LIN {X 0,Y 144.366,Z 912.436,A -85,B 0,C 180,E1 -24295.812,E2 -24295.812} C_VEL
LIN {X 0,Y 143.347,Z 905.875,A -85,B 0,C 180,E1 -24300,E2 -24300} C_VEL
LIN {X 0,Y 143.086,Z 898.213,A -85,B 0,C 180,E1 -24304.225,E2 -24304.225} C_VEL
LIN {X 0,Y 143.586,Z 889.005,A -85,B 0,C 180,E1 -24308.444,E2 -24308.444} C_VEL
LIN {X 0,Y 144.189,Z 880.732,A -85,B 0,C 180,E1 -24311.69,E2 -24311.69} C_VEL
LIN {X 0,Y 145.104,Z 871.718,A -85,B 0,C 180,E1 -24314.731,E2 -24314.731} C_VEL
LIN {X 0,Y 146.264,Z 860.917,A -85,B 0,C 180,E1 -24317.838,E2 -24317.838} C_VEL
LIN {X 0,Y 147.179,Z 852.291,A -85,B 0,C 180,E1 -24319.888,E2 -24319.888} C_VEL
LIN {X 0,Y 144.802,Z 841.839,A -85,B 0,C 180,E1 -24322.072,E2 -24322.072} C_VEL
LIN {X 0,Y 143.37,Z 834.62,A -85,B 0,C 180,E1 -24323.471,E2 -24323.471} C_VEL
LIN {X 0,Y 143.093,Z 834.654,A -85,B 0,C 180,E1 -24329.416,E2 -24329.416} C_VEL
LIN {X 0,Y 143.174,Z 834.808,A -85,B 0,C 180,E1 -24331.231,E2 -24331.231} C_VEL
LIN {X 0,Y 144.079,Z 837.334,A -85,B 0,C 180,E1 -24332.347,E2 -24332.347} C_VEL
LIN {X 0,Y 146.065,Z 839.541,A -85,B 0,C 180,E1 -24334.066,E2 -24334.066} C_VEL
LIN {X 0,Y 146.807,Z 840.16,A -85,B 0,C 180,E1 -24334.663,E2 -24334.663} C_VEL
LIN {X 0,Y 147.849,Z 842.508,A -85,B 0,C 180,E1 -24335.779,E2 -24335.779} C_VEL
LIN {X 0,Y 149.912,Z 845.217,A -85,B 0,C 180,E1 -24337.55,E2 -24337.55} C_VEL
LIN {X 0,Y 154.716,Z 853.873,A -85,B 0,C 180,E1 -24342.069,E2 -24342.069} C_VEL
LIN {X 0,Y 157.954,Z 860.834,A -85,B 0,C 180,E1 -24345.391,E2 -24345.391} C_VEL
LIN {X 0,Y 160.948,Z 868.94,A -85,B 0,C 180,E1 -24349.076,E2 -24349.076} C_VEL
LIN {X 0,Y 163.181,Z 877.591,A -85,B 0,C 180,E1 -24352.913,E2 -24352.913} C_VEL
LIN {X 0,Y 164.31,Z 884.842,A -85,B 0,C 180,E1 -24356.212,E2 -24356.212} C_VEL
LIN {X 0,Y 164.227,Z 886.502,A -85,B 0,C 180,E1 -24356.928,E2 -24356.928} C_VEL
LIN {X 0,Y 160.56,Z 894.538,A -85,B 0,C 180,E1 -24359.772,E2 -24359.772} C_VEL
LIN {X 0,Y 157.298,Z 901.182,A -85,B 0,C 180,E1 -24362.739,E2 -24362.739} C_VEL
LIN {X 0,Y 153.469,Z 908.642,A -85,B 0,C 180,E1 -24367.087,E2 -24367.087} C_VEL
LIN {X 0,Y 150.514,Z 913.635,A -85,B 0,C 180,E1 -24370.917,E2 -24370.917} C_VEL
LIN {X 0,Y 147.946,Z 917.527,A -85,B 0,C 180,E1 -24374.85,E2 -24374.85} C_VEL
LIN {X 0,Y 146.311,Z 920.348,A -85,B 0,C 180,E1 -24378.918,E2 -24378.918} C_VEL
LIN {X 0,Y 145.556,Z 921.691,A -85,B 0,C 180,E1 -24381.666,E2 -24381.666} C_VEL
LIN {X 0,Y 144.45,Z 923.269,A -85,B 0,C 180,E1 -24387.206,E2 -24387.206} C_VEL
LIN {X 0,Y 144.306,Z 923.495,A -85,B 0,C 180,E1 -24389.995,E2 -24389.995} C_VEL
LIN {X 0,Y 144.877,Z 922.719,A -85,B 0,C 180,E1 -24395.563,E2 -24395.563} C_VEL
LIN {X 0,Y 145.529,Z 921.77,A -85,B 0,C 180,E1 -24398.325,E2 -24398.325} C_VEL
LIN {X 0,Y 146.28,Z 920.46,A -85,B 0,C 180,E1 -24401.075,E2 -24401.075} C_VEL
LIN {X 0,Y 147.926,Z 917.671,A -85,B 0,C 180,E1 -24405.142,E2 -24405.142} C_VEL
LIN {X 0,Y 150.499,Z 913.82,A -85,B 0,C 180,E1 -24409.075,E2 -24409.075} C_VEL
LIN {X 0,Y 153.408,Z 908.893,A -85,B 0,C 180,E1 -24412.912,E2 -24412.912} C_VEL
LIN {X 0,Y 156.651,Z 902.704,A -85,B 0,C 180,E1 -24416.651,E2 -24416.651} C_VEL
LIN {X 0,Y 159.755,Z 896.388,A -85,B 0,C 180,E1 -24419.658,E2 -24419.658} C_VEL
LIN {X 0,Y 163.393,Z 888.72,A -85,B 0,C 180,E1 -24422.519,E2 -24422.519} C_VEL
LIN {X 0,Y 164.129,Z 886.977,A -85,B 0,C 180,E1 -24423.084,E2 -24423.084} C_VEL
LIN {X 0,Y 164.39,Z 885.314,A -85,B 0,C 180,E1 -24423.758,E2 -24423.758} C_VEL
LIN {X 0,Y 163.639,Z 879.851,A -85,B 0,C 180,E1 -24426.249,E2 -24426.249} C_VEL
LIN {X 0,Y 161.787,Z 871.808,A -85,B 0,C 180,E1 -24429.855,E2 -24429.855} C_VEL
LIN {X 0,Y 159.541,Z 864.62,A -85,B 0,C 180,E1 -24433.054,E2 -24433.054} C_VEL
LIN {X 0,Y 156.466,Z 857.156,A -85,B 0,C 180,E1 -24436.51,E2 -24436.51} C_VEL
LIN {X 0,Y 152.265,Z 848.934,A -85,B 0,C 180,E1 -24440.606,E2 -24440.606} C_VEL
LIN {X 0,Y 150.136,Z 845.542,A -85,B 0,C 180,E1 -24442.516,E2 -24442.516} C_VEL
LIN {X 0,Y 149.808,Z 844.719,A -85,B 0,C 180,E1 -24442.885,E2 -24442.885} C_VEL
LIN {X 0,Y 147.617,Z 841.995,A -85,B 0,C 180,E1 -24444.741,E2 -24444.741} C_VEL
LIN {X 0,Y 146.739,Z 839.962,A -85,B 0,C 180,E1 -24445.705,E2 -24445.705} C_VEL
LIN {X 0,Y 144.411,Z 837.842,A -85,B 0,C 180,E1 -24447.633,E2 -24447.633} C_VEL
LIN {X 0,Y 143.281,Z 835.366,A -85,B 0,C 180,E1 -24448.898,E2 -24448.898} C_VEL
LIN {X 0,Y 143.167,Z 834.643,A -85,B 0,C 180,E1 -24449.178,E2 -24449.178} C_VEL
LIN {X 0,Y 143.144,Z 834.646,A -85,B 0,C 180,E1 -24453.776,E2 -24453.776} C_VEL
LIN {X 0,Y 143.294,Z 834.627,A -85,B 0,C 180,E1 -24459.92,E2 -24459.92} C_VEL
LIN {X 0,Y 143.356,Z 834.615,A -85,B 0,C 180,E1 -24465.811,E2 -24465.811} C_VEL
LIN {X 0,Y 143.581,Z 834.6,A -85,B 0,C 180,E1 -24468.709,E2 -24468.709} C_VEL
LIN {X 0,Y 143.646,Z 834.581,A -85,B 0,C 180,E1 -24471.56,E2 -24471.56} C_VEL
LIN {X 0,Y 144.162,Z 834.535,A -85,B 0,C 180,E1 -24480,E2 -24480} C_VEL
LIN {X 0,Y 143.645,Z 834.591,A -85,B 0,C 180,E1 -24488.44,E2 -24488.44} C_VEL
LIN {X 0,Y 143.6,Z 834.597,A -85,B 0,C 180,E1 -24490.575,E2 -24490.575} C_VEL
LIN {X 0,Y 144.063,Z 838.083,A -85,B 0,C 180,E1 -24497.02,E2 -24497.02} C_VEL
LIN {X 0,Y 144.743,Z 841.753,A -85,B 0,C 180,E1 -24502.857,E2 -24502.857} C_VEL
LIN {X 0,Y 145.462,Z 844.863,A -85,B 0,C 180,E1 -24507.322,E2 -24507.322} C_VEL
LIN {X 0,Y 146.267,Z 848.468,A -85,B 0,C 180,E1 -24511.824,E2 -24511.824} C_VEL
LIN {X 0,Y 147.628,Z 851.95,A -85,B 0,C 180,E1 -24512.99,E2 -24512.99} C_VEL
LIN {X 0,Y 150.24,Z 856.036,A -85,B 0,C 180,E1 -24514.915,E2 -24514.915} C_VEL
LIN {X 0,Y 151.968,Z 860.121,A -85,B 0,C 180,E1 -24516.313,E2 -24516.313} C_VEL
LIN {X 0,Y 153.324,Z 862.543,A -85,B 0,C 180,E1 -24517.295,E2 -24517.295} C_VEL
LIN {X 0,Y 155.231,Z 867.069,A -85,B 0,C 180,E1 -24518.812,E2 -24518.812} C_VEL
LIN {X 0,Y 157.997,Z 874.12,A -85,B 0,C 180,E1 -24521.088,E2 -24521.088} C_VEL
LIN {X 0,Y 159.658,Z 879.116,A -85,B 0,C 180,E1 -24522.594,E2 -24522.594} C_VEL
LIN {X 0,Y 160.07,Z 883.691,A -85,B 0,C 180,E1 -24523.621,E2 -24523.621} C_VEL
LIN {X 0,Y 159.868,Z 895.589,A -85,B 0,C 180,E1 -24526.253,E2 -24526.253} C_VEL
LIN {X 0,Y 158.935,Z 906.349,A -85,B 0,C 180,E1 -24528.914,E2 -24528.914} C_VEL
LIN {X 0,Y 157.059,Z 917.445,A -85,B 0,C 180,E1 -24532.034,E2 -24532.034} C_VEL
LIN {X 0,Y 154.947,Z 926.905,A -85,B 0,C 180,E1 -24535.196,E2 -24535.196} C_VEL
LIN {X 0,Y 152.285,Z 935.787,A -85,B 0,C 180,E1 -24538.728,E2 -24538.728} C_VEL
LIN {X 0,Y 149.406,Z 943.829,A -85,B 0,C 180,E1 -24542.707,E2 -24542.707} C_VEL
LIN {X 0,Y 146.757,Z 949.26,A -85,B 0,C 180,E1 -24545.986,E2 -24545.986} C_VEL
LIN {X 0,Y 144.349,Z 954.58,A -85,B 0,C 180,E1 -24550.079,E2 -24550.079} C_VEL
LIN {X 0,Y 142.88,Z 958.794,A -85,B 0,C 180,E1 -24554.309,E2 -24554.309} C_VEL
LIN {X 0,Y 142.204,Z 961.975,A -85,B 0,C 180,E1 -24558.604,E2 -24558.604} C_VEL
LIN {X 0,Y 142.218,Z 963.539,A -85,B 0,C 180,E1 -24561.48,E2 -24561.48} C_VEL
LIN {X 0,Y 142.458,Z 964.687,A -85,B 0,C 180,E1 -24564.343,E2 -24564.343} C_VEL
LIN {X 0,Y 142.828,Z 965.417,A -85,B 0,C 180,E1 -24567.185,E2 -24567.185} C_VEL
LIN {X 0,Y 143.31,Z 965.72,A -85,B 0,C 180,E1 -24570.005,E2 -24570.005} C_VEL
LIN {X 0,Y 142.839,Z 965.402,A -85,B 0,C 180,E1 -24572.825,E2 -24572.825} C_VEL
LIN {X 0,Y 142.47,Z 964.661,A -85,B 0,C 180,E1 -24575.667,E2 -24575.667} C_VEL
LIN {X 0,Y 142.254,Z 963.362,A -85,B 0,C 180,E1 -24578.85,E2 -24578.85} C_VEL
LIN {X 0,Y 142.808,Z 959.914,A -85,B 0,C 180,E1 -24584.25,E2 -24584.25} C_VEL
LIN {X 0,Y 144.374,Z 956.094,A -85,B 0,C 180,E1 -24588.451,E2 -24588.451} C_VEL
LIN {X 0,Y 145.697,Z 953.524,A -85,B 0,C 180,E1 -24590.844,E2 -24590.844} C_VEL
LIN {X 0,Y 150.579,Z 952.693,A -85,B 0,C 180,E1 -24597.827,E2 -24597.827} C_VEL
LIN {X 0,Y 156.123,Z 950.986,A -85,B 0,C 180,E1 -24602.702,E2 -24602.702} C_VEL
LIN {X 0,Y 162.654,Z 948.312,A -85,B 0,C 180,E1 -24607.228,E2 -24607.228} C_VEL
LIN {X 0,Y 172.423,Z 943.736,A -85,B 0,C 180,E1 -24612.269,E2 -24612.269} C_VEL
LIN {X 0,Y 180.891,Z 939.233,A -85,B 0,C 180,E1 -24615.982,E2 -24615.982} C_VEL
LIN {X 0,Y 191.252,Z 932.914,A -85,B 0,C 180,E1 -24620.511,E2 -24620.511} C_VEL
LIN {X 0,Y 191.517,Z 932.705,A -85,B 0,C 180,E1 -24620.717,E2 -24620.717} C_VEL
LIN {X 0,Y 191.421,Z 932.464,A -85,B 0,C 180,E1 -24621.257,E2 -24621.257} C_VEL
LIN {X 0,Y 190.034,Z 932.668,A -85,B 0,C 180,E1 -24621.886,E2 -24621.886} C_VEL
LIN {X 0,Y 186.966,Z 933.43,A -85,B 0,C 180,E1 -24622.572,E2 -24622.572} C_VEL
LIN {X 0,Y 178.48,Z 935.34,A -85,B 0,C 180,E1 -24623.75,E2 -24623.75} C_VEL
LIN {X 0,Y 174.831,Z 935.868,A -85,B 0,C 180,E1 -24624.643,E2 -24624.643} C_VEL
LIN {X 0,Y 174.697,Z 935.77,A -85,B 0,C 180,E1 -24624.691,E2 -24624.691} C_VEL
LIN {X 0,Y 168.525,Z 935.804,A -85,B 0,C 180,E1 -24627.171,E2 -24627.171} C_VEL
LIN {X 0,Y 160.286,Z 934.779,A -85,B 0,C 180,E1 -24631.163,E2 -24631.163} C_VEL
LIN {X 0,Y 153.031,Z 932.451,A -85,B 0,C 180,E1 -24635.586,E2 -24635.586} C_VEL
LIN {X 0,Y 146.958,Z 928.79,A -85,B 0,C 180,E1 -24640.442,E2 -24640.442} C_VEL
LIN {X 0,Y 143.316,Z 925.246,A -85,B 0,C 180,E1 -24644.353,E2 -24644.353} C_VEL
LIN {X 0,Y 139.704,Z 919.181,A -85,B 0,C 180,E1 -24649.859,E2 -24649.859} C_VEL
LIN {X 0,Y 137.797,Z 913.654,A -85,B 0,C 180,E1 -24654.145,E2 -24654.145} C_VEL
LIN {X 0,Y 136.476,Z 907.094,A -85,B 0,C 180,E1 -24658.525,E2 -24658.525} C_VEL
LIN {X 0,Y 136.065,Z 899.483,A -85,B 0,C 180,E1 -24662.961,E2 -24662.961} C_VEL
LIN {X 0,Y 136.364,Z 890.328,A -85,B 0,C 180,E1 -24667.403,E2 -24667.403} C_VEL
LIN {X 0,Y 136.912,Z 883.366,A -85,B 0,C 180,E1 -24670.35,E2 -24670.35} C_VEL
LIN {X 0,Y 137.771,Z 873.83,A -85,B 0,C 180,E1 -24673.826,E2 -24673.826} C_VEL
LIN {X 0,Y 138.966,Z 862.632,A -85,B 0,C 180,E1 -24677.285,E2 -24677.285} C_VEL
LIN {X 0,Y 140.022,Z 852.636,A -85,B 0,C 180,E1 -24679.804,E2 -24679.804} C_VEL
LIN {X 0,Y 137.087,Z 839.359,A -85,B 0,C 180,E1 -24682.649,E2 -24682.649} C_VEL
LIN {X 0,Y 136.33,Z 835.495,A -85,B 0,C 180,E1 -24683.37,E2 -24683.37} C_VEL
LIN {X 0,Y 136.151,Z 835.514,A -85,B 0,C 180,E1 -24685.615,E2 -24685.615} C_VEL
LIN {X 0,Y 136.777,Z 837.767,A -85,B 0,C 180,E1 -24686.718,E2 -24686.718} C_VEL
LIN {X 0,Y 138.807,Z 840.306,A -85,B 0,C 180,E1 -24689.042,E2 -24689.042} C_VEL
LIN {X 0,Y 140.121,Z 841.306,A -85,B 0,C 180,E1 -24690.312,E2 -24690.312} C_VEL
LIN {X 0,Y 141.683,Z 844.429,A -85,B 0,C 180,E1 -24692.225,E2 -24692.225} C_VEL
LIN {X 0,Y 143.674,Z 846.973,A -85,B 0,C 180,E1 -24694.23,E2 -24694.23} C_VEL
LIN {X 0,Y 148.124,Z 854.661,A -85,B 0,C 180,E1 -24698.952,E2 -24698.952} C_VEL
LIN {X 0,Y 151.725,Z 862.39,A -85,B 0,C 180,E1 -24703.096,E2 -24703.096} C_VEL
LIN {X 0,Y 154.623,Z 870.194,A -85,B 0,C 180,E1 -24707.011,E2 -24707.011} C_VEL
LIN {X 0,Y 156.635,Z 877.883,A -85,B 0,C 180,E1 -24710.714,E2 -24710.714} C_VEL
LIN {X 0,Y 157.81,Z 884.685,A -85,B 0,C 180,E1 -24714.031,E2 -24714.031} C_VEL
LIN {X 0,Y 158.1,Z 887.587,A -85,B 0,C 180,E1 -24715.47,E2 -24715.47} C_VEL
LIN {X 0,Y 157.682,Z 889.267,A -85,B 0,C 180,E1 -24716.137,E2 -24716.137} C_VEL
LIN {X 0,Y 153.771,Z 897.031,A -85,B 0,C 180,E1 -24719.053,E2 -24719.053} C_VEL
LIN {X 0,Y 149.84,Z 904.624,A -85,B 0,C 180,E1 -24722.833,E2 -24722.833} C_VEL
LIN {X 0,Y 145.987,Z 911.438,A -85,B 0,C 180,E1 -24727.343,E2 -24727.343} C_VEL
LIN {X 0,Y 142.858,Z 916.073,A -85,B 0,C 180,E1 -24731.346,E2 -24731.346} C_VEL
LIN {X 0,Y 140.473,Z 919.593,A -85,B 0,C 180,E1 -24735.508,E2 -24735.508} C_VEL
LIN {X 0,Y 139.425,Z 921.38,A -85,B 0,C 180,E1 -24738.363,E2 -24738.363} C_VEL
LIN {X 0,Y 138.609,Z 922.722,A -85,B 0,C 180,E1 -24741.246,E2 -24741.246} C_VEL
LIN {X 0,Y 137.435,Z 924.3,A -85,B 0,C 180,E1 -24747.064,E2 -24747.064} C_VEL
LIN {X 0,Y 137.281,Z 924.526,A -85,B 0,C 180,E1 -24749.995,E2 -24749.995} C_VEL
LIN {X 0,Y 137.888,Z 923.75,A -85,B 0,C 180,E1 -24755.845,E2 -24755.845} C_VEL
LIN {X 0,Y 138.584,Z 922.8,A -85,B 0,C 180,E1 -24758.745,E2 -24758.745} C_VEL
LIN {X 0,Y 139.396,Z 921.491,A -85,B 0,C 180,E1 -24761.629,E2 -24761.629} C_VEL
LIN {X 0,Y 141.156,Z 918.702,A -85,B 0,C 180,E1 -24765.887,E2 -24765.887} C_VEL
LIN {X 0,Y 143.878,Z 914.851,A -85,B 0,C 180,E1 -24769.989,E2 -24769.989} C_VEL
LIN {X 0,Y 146.972,Z 909.922,A -85,B 0,C 180,E1 -24773.977,E2 -24773.977} C_VEL
LIN {X 0,Y 150.406,Z 903.734,A -85,B 0,C 180,E1 -24777.851,E2 -24777.851} C_VEL
LIN {X 0,Y 153.69,Z 897.416,A -85,B 0,C 180,E1 -24780.954,E2 -24780.954} C_VEL
LIN {X 0,Y 157.537,Z 889.745,A -85,B 0,C 180,E1 -24783.887,E2 -24783.887} C_VEL
LIN {X 0,Y 158.133,Z 888.033,A -85,B 0,C 180,E1 -24784.511,E2 -24784.511} C_VEL
LIN {X 0,Y 157.366,Z 881.445,A -85,B 0,C 180,E1 -24787.757,E2 -24787.757} C_VEL
LIN {X 0,Y 155.957,Z 874.774,A -85,B 0,C 180,E1 -24790.991,E2 -24790.991} C_VEL
LIN {X 0,Y 153.883,Z 867.701,A -85,B 0,C 180,E1 -24794.399,E2 -24794.399} C_VEL
LIN {X 0,Y 150.987,Z 860.341,A -85,B 0,C 180,E1 -24798.13,E2 -24798.13} C_VEL
LIN {X 0,Y 147.718,Z 853.794,A -85,B 0,C 180,E1 -24801.793,E2 -24801.793} C_VEL
LIN {X 0,Y 145.929,Z 850.339,A -85,B 0,C 180,E1 -24803.769,E2 -24803.769} C_VEL
LIN {X 0,Y 143.891,Z 847.331,A -85,B 0,C 180,E1 -24805.829,E2 -24805.829} C_VEL
LIN {X 0,Y 143.495,Z 846.305,A -85,B 0,C 180,E1 -24806.358,E2 -24806.358} C_VEL
LIN {X 0,Y 140.627,Z 842.66,A -85,B 0,C 180,E1 -24809.29,E2 -24809.29} C_VEL
LIN {X 0,Y 139.947,Z 840.995,A -85,B 0,C 180,E1 -24810.232,E2 -24810.232} C_VEL
LIN {X 0,Y 137.43,Z 838.858,A -85,B 0,C 180,E1 -24812.803,E2 -24812.803} C_VEL
LIN {X 0,Y 136.28,Z 836.54,A -85,B 0,C 180,E1 -24814.411,E2 -24814.411} C_VEL
LIN {X 0,Y 136.076,Z 835.525,A -85,B 0,C 180,E1 -24814.882,E2 -24814.882} C_VEL
LIN {X 0,Y 136.231,Z 835.506,A -85,B 0,C 180,E1 -24818.831,E2 -24818.831} C_VEL
LIN {X 0,Y 136.262,Z 835.495,A -85,B 0,C 180,E1 -24825.055,E2 -24825.055} C_VEL
LIN {X 0,Y 136.484,Z 835.487,A -85,B 0,C 180,E1 -24828.113,E2 -24828.113} C_VEL
LIN {X 0,Y 136.574,Z 835.461,A -85,B 0,C 180,E1 -24831.119,E2 -24831.119} C_VEL
LIN {X 0,Y 137.119,Z 835.412,A -85,B 0,C 180,E1 -24840,E2 -24840} C_VEL
LIN {X 0,Y 136.564,Z 835.579,A -85,B 0,C 180,E1 -24847.392,E2 -24847.392} C_VEL
LIN {X 0,Y 136.957,Z 838.124,A -85,B 0,C 180,E1 -24852.869,E2 -24852.869} C_VEL
LIN {X 0,Y 137.38,Z 840.825,A -85,B 0,C 180,E1 -24857.875,E2 -24857.875} C_VEL
LIN {X 0,Y 138.164,Z 844.553,A -85,B 0,C 180,E1 -24864.013,E2 -24864.013} C_VEL
LIN {X 0,Y 138.48,Z 846.05,A -85,B 0,C 180,E1 -24866.161,E2 -24866.161} C_VEL
LIN {X 0,Y 140.057,Z 849.793,A -85,B 0,C 180,E1 -24867.859,E2 -24867.859} C_VEL
LIN {X 0,Y 143.028,Z 854.216,A -85,B 0,C 180,E1 -24870.548,E2 -24870.548} C_VEL
LIN {X 0,Y 144.665,Z 858.223,A -85,B 0,C 180,E1 -24872.168,E2 -24872.168} C_VEL
LIN {X 0,Y 146.467,Z 861.341,A -85,B 0,C 180,E1 -24873.698,E2 -24873.698} C_VEL
LIN {X 0,Y 148.558,Z 866.21,A -85,B 0,C 180,E1 -24875.625,E2 -24875.625} C_VEL
LIN {X 0,Y 151.111,Z 872.345,A -85,B 0,C 180,E1 -24877.957,E2 -24877.957} C_VEL
LIN {X 0,Y 154.309,Z 882.048,A -85,B 0,C 180,E1 -24881.24,E2 -24881.24} C_VEL
LIN {X 0,Y 154.536,Z 886.531,A -85,B 0,C 180,E1 -24882.346,E2 -24882.346} C_VEL
LIN {X 0,Y 153.922,Z 898.527,A -85,B 0,C 180,E1 -24885.229,E2 -24885.229} C_VEL
LIN {X 0,Y 152.495,Z 909.51,A -85,B 0,C 180,E1 -24888.2,E2 -24888.2} C_VEL
LIN {X 0,Y 150.426,Z 919.596,A -85,B 0,C 180,E1 -24891.333,E2 -24891.333} C_VEL
LIN {X 0,Y 148.051,Z 928.69,A -85,B 0,C 180,E1 -24894.679,E2 -24894.679} C_VEL
LIN {X 0,Y 145.031,Z 937.582,A -85,B 0,C 180,E1 -24898.612,E2 -24898.612} C_VEL
LIN {X 0,Y 142.471,Z 943.932,A -85,B 0,C 180,E1 -24902.061,E2 -24902.061} C_VEL
LIN {X 0,Y 139.262,Z 950.097,A -85,B 0,C 180,E1 -24906.195,E2 -24906.195} C_VEL
LIN {X 0,Y 136.979,Z 955.041,A -85,B 0,C 180,E1 -24910.525,E2 -24910.525} C_VEL
LIN {X 0,Y 135.624,Z 958.897,A -85,B 0,C 180,E1 -24914.989,E2 -24914.989} C_VEL
LIN {X 0,Y 135.202,Z 960.926,A -85,B 0,C 180,E1 -24918.005,E2 -24918.005} C_VEL
LIN {X 0,Y 135.166,Z 962.514,A -85,B 0,C 180,E1 -24921.082,E2 -24921.082} C_VEL
LIN {X 0,Y 135.387,Z 963.644,A -85,B 0,C 180,E1 -24924.046,E2 -24924.046} C_VEL
LIN {X 0,Y 135.749,Z 964.377,A -85,B 0,C 180,E1 -24927.038,E2 -24927.038} C_VEL
LIN {X 0,Y 136.252,Z 964.684,A -85,B 0,C 180,E1 -24930.005,E2 -24930.005} C_VEL
LIN {X 0,Y 135.761,Z 964.362,A -85,B 0,C 180,E1 -24932.973,E2 -24932.973} C_VEL
LIN {X 0,Y 135.403,Z 963.618,A -85,B 0,C 180,E1 -24935.964,E2 -24935.964} C_VEL
LIN {X 0,Y 135.216,Z 962.427,A -85,B 0,C 180,E1 -24939.052,E2 -24939.052} C_VEL
LIN {X 0,Y 135.572,Z 959.919,A -85,B 0,C 180,E1 -24943.495,E2 -24943.495} C_VEL
LIN {X 0,Y 136.971,Z 956.433,A -85,B 0,C 180,E1 -24947.936,E2 -24947.936} C_VEL
LIN {X 0,Y 139.62,Z 951.559,A -85,B 0,C 180,E1 -24952.576,E2 -24952.576} C_VEL
LIN {X 0,Y 144.419,Z 951.135,A -85,B 0,C 180,E1 -24959.125,E2 -24959.125} C_VEL
LIN {X 0,Y 150.223,Z 949.812,A -85,B 0,C 180,E1 -24964.158,E2 -24964.158} C_VEL
LIN {X 0,Y 157.04,Z 947.521,A -85,B 0,C 180,E1 -24968.8,E2 -24968.8} C_VEL
LIN {X 0,Y 165.04,Z 944.315,A -85,B 0,C 180,E1 -24972.953,E2 -24972.953} C_VEL
LIN {X 0,Y 172.589,Z 941.071,A -85,B 0,C 180,E1 -24976.191,E2 -24976.191} C_VEL
LIN {X 0,Y 182.399,Z 936.056,A -85,B 0,C 180,E1 -24980.415,E2 -24980.415} C_VEL
LIN {X 0,Y 183.903,Z 934.973,A -85,B 0,C 180,E1 -24981.557,E2 -24981.557} C_VEL
LIN {X 0,Y 174.697,Z 935.77,A -85,B 0,C 180,E1 -24984.691,E2 -24984.691} C_VEL
LIN {X 0,Y 170.39,Z 936.029,A -85,B 0,C 180,E1 -24986.034,E2 -24986.034} C_VEL
LIN {X 0,Y 162.285,Z 936.266,A -85,B 0,C 180,E1 -24987.999,E2 -24987.999} C_VEL
LIN {X 0,Y 154.466,Z 935.642,A -85,B 0,C 180,E1 -24990.169,E2 -24990.169} C_VEL
LIN {X 0,Y 150.695,Z 934.721,A -85,B 0,C 180,E1 -24991.837,E2 -24991.837} C_VEL
LIN {X 0,Y 143.285,Z 931.186,A -85,B 0,C 180,E1 -24996.897,E2 -24996.897} C_VEL
LIN {X 0,Y 137.63,Z 926.44,A -85,B 0,C 180,E1 -25002.158,E2 -25002.158} C_VEL
LIN {X 0,Y 133.53,Z 920.33,A -85,B 0,C 180,E1 -25007.847,E2 -25007.847} C_VEL
LIN {X 0,Y 131.397,Z 914.79,A -85,B 0,C 180,E1 -25012.316,E2 -25012.316} C_VEL
LIN {X 0,Y 129.779,Z 908.229,A -85,B 0,C 180,E1 -25016.896,E2 -25016.896} C_VEL
LIN {X 0,Y 129.155,Z 900.655,A -85,B 0,C 180,E1 -25021.559,E2 -25021.559} C_VEL
LIN {X 0,Y 129.173,Z 891.522,A -85,B 0,C 180,E1 -25026.247,E2 -25026.247} C_VEL
LIN {X 0,Y 129.736,Z 884.648,A -85,B 0,C 180,E1 -25029.353,E2 -25029.353} C_VEL
LIN {X 0,Y 130.456,Z 875.609,A -85,B 0,C 180,E1 -25032.88,E2 -25032.88} C_VEL
LIN {X 0,Y 131.672,Z 864.16,A -85,B 0,C 180,E1 -25036.672,E2 -25036.672} C_VEL
LIN {X 0,Y 132.866,Z 852.817,A -85,B 0,C 180,E1 -25039.707,E2 -25039.707} C_VEL
LIN {X 0,Y 130.692,Z 843.478,A -85,B 0,C 180,E1 -25041.905,E2 -25041.905} C_VEL
LIN {X 0,Y 131.038,Z 844.373,A -85,B 0,C 180,E1 -25042.631,E2 -25042.631} C_VEL
LIN {X 0,Y 132.27,Z 844.06,A -85,B 0,C 180,E1 -25043.929,E2 -25043.929} C_VEL
LIN {X 0,Y 133.601,Z 842.617,A -85,B 0,C 180,E1 -25044.888,E2 -25044.888} C_VEL
LIN {X 0,Y 134.845,Z 845.291,A -85,B 0,C 180,E1 -25046.923,E2 -25046.923} C_VEL
LIN {X 0,Y 136.571,Z 847.068,A -85,B 0,C 180,E1 -25048.966,E2 -25048.966} C_VEL
LIN {X 0,Y 140.11,Z 852.88,A -85,B 0,C 180,E1 -25053.489,E2 -25053.489} C_VEL
LIN {X 0,Y 143.612,Z 859.568,A -85,B 0,C 180,E1 -25057.892,E2 -25057.892} C_VEL
LIN {X 0,Y 146.695,Z 866.756,A -85,B 0,C 180,E1 -25062.123,E2 -25062.123} C_VEL
LIN {X 0,Y 149.263,Z 874.433,A -85,B 0,C 180,E1 -25066.31,E2 -25066.31} C_VEL
LIN {X 0,Y 150.916,Z 881.903,A -85,B 0,C 180,E1 -25070.208,E2 -25070.208} C_VEL
LIN {X 0,Y 151.8,Z 888.725,A -85,B 0,C 180,E1 -25073.817,E2 -25073.817} C_VEL
LIN {X 0,Y 151.824,Z 890.315,A -85,B 0,C 180,E1 -25074.641,E2 -25074.641} C_VEL
LIN {X 0,Y 147.796,Z 898.064,A -85,B 0,C 180,E1 -25077.654,E2 -25077.654} C_VEL
LIN {X 0,Y 143.629,Z 905.651,A -85,B 0,C 180,E1 -25081.549,E2 -25081.549} C_VEL
LIN {X 0,Y 139.534,Z 912.47,A -85,B 0,C 180,E1 -25086.233,E2 -25086.233} C_VEL
LIN {X 0,Y 136.222,Z 917.106,A -85,B 0,C 180,E1 -25090.401,E2 -25090.401} C_VEL
LIN {X 0,Y 133.683,Z 920.625,A -85,B 0,C 180,E1 -25094.755,E2 -25094.755} C_VEL
LIN {X 0,Y 132.552,Z 922.412,A -85,B 0,C 180,E1 -25097.75,E2 -25097.75} C_VEL
LIN {X 0,Y 131.671,Z 923.754,A -85,B 0,C 180,E1 -25100.78,E2 -25100.78} C_VEL
LIN {X 0,Y 130.421,Z 925.331,A -85,B 0,C 180,E1 -25106.906,E2 -25106.906} C_VEL
LIN {X 0,Y 130.279,Z 925.554,A -85,B 0,C 180,E1 -25109.994,E2 -25109.994} C_VEL
LIN {X 0,Y 130.902,Z 924.781,A -85,B 0,C 180,E1 -25116.159,E2 -25116.159} C_VEL
LIN {X 0,Y 131.647,Z 923.831,A -85,B 0,C 180,E1 -25119.21,E2 -25119.21} C_VEL
LIN {X 0,Y 132.526,Z 922.521,A -85,B 0,C 180,E1 -25122.241,E2 -25122.241} C_VEL
LIN {X 0,Y 134.413,Z 919.732,A -85,B 0,C 180,E1 -25126.707,E2 -25126.707} C_VEL
LIN {X 0,Y 137.297,Z 915.881,A -85,B 0,C 180,E1 -25130.991,E2 -25130.991} C_VEL
LIN {X 0,Y 140.592,Z 910.95,A -85,B 0,C 180,E1 -25135.138,E2 -25135.138} C_VEL
LIN {X 0,Y 144.254,Z 904.759,A -85,B 0,C 180,E1 -25139.15,E2 -25139.15} C_VEL
LIN {X 0,Y 147.711,Z 898.445,A -85,B 0,C 180,E1 -25142.356,E2 -25142.356} C_VEL
LIN {X 0,Y 151.754,Z 890.773,A -85,B 0,C 180,E1 -25145.367,E2 -25145.367} C_VEL
LIN {X 0,Y 151.779,Z 887.577,A -85,B 0,C 180,E1 -25147.003,E2 -25147.003} C_VEL
LIN {X 0,Y 150.718,Z 880.484,A -85,B 0,C 180,E1 -25150.748,E2 -25150.748} C_VEL
LIN {X 0,Y 149.242,Z 874.037,A -85,B 0,C 180,E1 -25154.098,E2 -25154.098} C_VEL
LIN {X 0,Y 146.922,Z 866.929,A -85,B 0,C 180,E1 -25157.956,E2 -25157.956} C_VEL
LIN {X 0,Y 143.859,Z 859.73,A -85,B 0,C 180,E1 -25162.185,E2 -25162.185} C_VEL
LIN {X 0,Y 141.858,Z 855.773,A -85,B 0,C 180,E1 -25164.728,E2 -25164.728} C_VEL
LIN {X 0,Y 139.201,Z 851.33,A -85,B 0,C 180,E1 -25167.986,E2 -25167.986} C_VEL
LIN {X 0,Y 137.194,Z 848.057,A -85,B 0,C 180,E1 -25170.546,E2 -25170.546} C_VEL
LIN {X 0,Y 134.038,Z 843.876,A -85,B 0,C 180,E1 -25174.681,E2 -25174.681} C_VEL
LIN {X 0,Y 133.377,Z 842.096,A -85,B 0,C 180,E1 -25175.897,E2 -25175.897} C_VEL
LIN {X 0,Y 130.664,Z 839.968,A -85,B 0,C 180,E1 -25179.742,E2 -25179.742} C_VEL
LIN {X 0,Y 129.475,Z 837.71,A -85,B 0,C 180,E1 -25182.12,E2 -25182.12} C_VEL
LIN {X 0,Y 129.169,Z 836.385,A -85,B 0,C 180,E1 -25183.097,E2 -25183.097} C_VEL
LIN {X 0,Y 129.403,Z 836.37,A -85,B 0,C 180,E1 -25187.819,E2 -25187.819} C_VEL
LIN {X 0,Y 129.501,Z 836.341,A -85,B 0,C 180,E1 -25190.63,E2 -25190.63} C_VEL
LIN {X 0,Y 130.074,Z 836.29,A -85,B 0,C 180,E1 -25200,E2 -25200} C_VEL
LIN {X 0,Y 129.668,Z 836.369,A -85,B 0,C 180,E1 -25203.107,E2 -25203.107} C_VEL
LIN {X 0,Y 130.044,Z 838.775,A -85,B 0,C 180,E1 -25209.33,E2 -25209.33} C_VEL
LIN {X 0,Y 130.284,Z 840.911,A -85,B 0,C 180,E1 -25213.863,E2 -25213.863} C_VEL
LIN {X 0,Y 130.676,Z 843.232,A -85,B 0,C 180,E1 -25218.014,E2 -25218.014} C_VEL
LIN {X 0,Y 132.152,Z 846.897,A -85,B 0,C 180,E1 -25220.426,E2 -25220.426} C_VEL
LIN {X 0,Y 135.604,Z 851.784,A -85,B 0,C 180,E1 -25224.699,E2 -25224.699} C_VEL
LIN {X 0,Y 137.658,Z 856.523,A -85,B 0,C 180,E1 -25227.251,E2 -25227.251} C_VEL
LIN {X 0,Y 139.619,Z 859.82,A -85,B 0,C 180,E1 -25229.289,E2 -25229.289} C_VEL
LIN {X 0,Y 141.505,Z 864.406,A -85,B 0,C 180,E1 -25231.432,E2 -25231.432} C_VEL
LIN {X 0,Y 142.582,Z 866.601,A -85,B 0,C 180,E1 -25232.519,E2 -25232.519} C_VEL
LIN {X 0,Y 145.688,Z 874.975,A -85,B 0,C 180,E1 -25235.993,E2 -25235.993} C_VEL
LIN {X 0,Y 148.16,Z 882.618,A -85,B 0,C 180,E1 -25238.942,E2 -25238.942} C_VEL
LIN {X 0,Y 149.004,Z 885.622,A -85,B 0,C 180,E1 -25240.035,E2 -25240.035} C_VEL
LIN {X 0,Y 148.927,Z 890.7,A -85,B 0,C 180,E1 -25241.351,E2 -25241.351} C_VEL
LIN {X 0,Y 147.795,Z 902.565,A -85,B 0,C 180,E1 -25244.505,E2 -25244.505} C_VEL
LIN {X 0,Y 145.925,Z 912.96,A -85,B 0,C 180,E1 -25247.61,E2 -25247.61} C_VEL
LIN {X 0,Y 143.132,Z 923.887,A -85,B 0,C 180,E1 -25251.446,E2 -25251.446} C_VEL
LIN {X 0,Y 140.471,Z 932.069,A -85,B 0,C 180,E1 -25254.882,E2 -25254.882} C_VEL
LIN {X 0,Y 137.197,Z 940.485,A -85,B 0,C 180,E1 -25259.192,E2 -25259.192} C_VEL
LIN {X 0,Y 134.963,Z 945.088,A -85,B 0,C 180,E1 -25262.059,E2 -25262.059} C_VEL
LIN {X 0,Y 131.774,Z 950.809,A -85,B 0,C 180,E1 -25266.428,E2 -25266.428} C_VEL
LIN {X 0,Y 129.612,Z 955.379,A -85,B 0,C 180,E1 -25271.02,E2 -25271.02} C_VEL
LIN {X 0,Y 128.405,Z 958.899,A -85,B 0,C 180,E1 -25275.747,E2 -25275.747} C_VEL
LIN {X 0,Y 128.106,Z 961.604,A -85,B 0,C 180,E1 -25280.93,E2 -25280.93} C_VEL
LIN {X 0,Y 128.298,Z 962.598,A -85,B 0,C 180,E1 -25283.716,E2 -25283.716} C_VEL
LIN {X 0,Y 128.673,Z 963.336,A -85,B 0,C 180,E1 -25286.875,E2 -25286.875} C_VEL
LIN {X 0,Y 129.191,Z 963.647,A -85,B 0,C 180,E1 -25290.006,E2 -25290.006} C_VEL
LIN {X 0,Y 128.684,Z 963.321,A -85,B 0,C 180,E1 -25293.136,E2 -25293.136} C_VEL
LIN {X 0,Y 128.318,Z 962.572,A -85,B 0,C 180,E1 -25296.294,E2 -25296.294} C_VEL
LIN {X 0,Y 128.159,Z 961.41,A -85,B 0,C 180,E1 -25299.475,E2 -25299.475} C_VEL
LIN {X 0,Y 128.656,Z 958.873,A -85,B 0,C 180,E1 -25304.236,E2 -25304.236} C_VEL
LIN {X 0,Y 130.211,Z 955.386,A -85,B 0,C 180,E1 -25308.901,E2 -25308.901} C_VEL
LIN {X 0,Y 133.341,Z 950.027,A -85,B 0,C 180,E1 -25314.115,E2 -25314.115} C_VEL
LIN {X 0,Y 133.758,Z 949.562,A -85,B 0,C 180,E1 -25314.654,E2 -25314.654} C_VEL
LIN {X 0,Y 137.628,Z 949.533,A -85,B 0,C 180,E1 -25319.761,E2 -25319.761} C_VEL
LIN {X 0,Y 144.454,Z 948.485,A -85,B 0,C 180,E1 -25325.726,E2 -25325.726} C_VEL
LIN {X 0,Y 151.57,Z 946.558,A -85,B 0,C 180,E1 -25330.483,E2 -25330.483} C_VEL
LIN {X 0,Y 159.908,Z 943.863,A -85,B 0,C 180,E1 -25334.69,E2 -25334.69} C_VEL
LIN {X 0,Y 168.924,Z 940.342,A -85,B 0,C 180,E1 -25338.499,E2 -25338.499} C_VEL
LIN {X 0,Y 174.309,Z 937.959,A -85,B 0,C 180,E1 -25340.769,E2 -25340.769} C_VEL
LIN {X 0,Y 174.866,Z 937.484,A -85,B 0,C 180,E1 -25341.391,E2 -25341.391} C_VEL
LIN {X 0,Y 162.724,Z 937.319,A -85,B 0,C 180,E1 -25345.843,E2 -25345.843} C_VEL
LIN {X 0,Y 154.172,Z 935.791,A -85,B 0,C 180,E1 -25349.905,E2 -25349.905} C_VEL
LIN {X 0,Y 150.695,Z 934.721,A -85,B 0,C 180,E1 -25351.837,E2 -25351.837} C_VEL
LIN {X 0,Y 147.081,Z 933.617,A -85,B 0,C 180,E1 -25353.586,E2 -25353.586} C_VEL
LIN {X 0,Y 140.102,Z 931.311,A -85,B 0,C 180,E1 -25356.241,E2 -25356.241} C_VEL
LIN {X 0,Y 133.627,Z 928.39,A -85,B 0,C 180,E1 -25359.118,E2 -25359.118} C_VEL
LIN {X 0,Y 130.906,Z 926.167,A -85,B 0,C 180,E1 -25361.191,E2 -25361.191} C_VEL
LIN {X 0,Y 126.638,Z 919.689,A -85,B 0,C 180,E1 -25367.174,E2 -25367.174} C_VEL
LIN {X 0,Y 123.76,Z 911.666,A -85,B 0,C 180,E1 -25373.479,E2 -25373.479} C_VEL
LIN {X 0,Y 122.277,Z 901.709,A -85,B 0,C 180,E1 -25380,E2 -25380} C_VEL
LIN {X 0,Y 122.122,Z 892.616,A -85,B 0,C 180,E1 -25384.952,E2 -25384.952} C_VEL
LIN {X 0,Y 122.723,Z 883.928,A -85,B 0,C 180,E1 -25389.061,E2 -25389.061} C_VEL
LIN {X 0,Y 123.533,Z 873.703,A -85,B 0,C 180,E1 -25393.154,E2 -25393.154} C_VEL
LIN {X 0,Y 124.83,Z 861.604,A -85,B 0,C 180,E1 -25397.191,E2 -25397.191} C_VEL
LIN {X 0,Y 125.65,Z 853.572,A -85,B 0,C 180,E1 -25399.396,E2 -25399.396} C_VEL
LIN {X 0,Y 125.652,Z 853.946,A -85,B 0,C 180,E1 -25399.609,E2 -25399.609} C_VEL
LIN {X 0,Y 128.136,Z 853.05,A -85,B 0,C 180,E1 -25402.578,E2 -25402.578} C_VEL
LIN {X 0,Y 129.969,Z 851.096,A -85,B 0,C 180,E1 -25403.926,E2 -25403.926} C_VEL
LIN {X 0,Y 131.423,Z 850.61,A -85,B 0,C 180,E1 -25405.329,E2 -25405.329} C_VEL
LIN {X 0,Y 133.451,Z 853.268,A -85,B 0,C 180,E1 -25408.293,E2 -25408.293} C_VEL
LIN {X 0,Y 136.815,Z 859.808,A -85,B 0,C 180,E1 -25413.519,E2 -25413.519} C_VEL
LIN {X 0,Y 139.835,Z 866.289,A -85,B 0,C 180,E1 -25418.088,E2 -25418.088} C_VEL
LIN {X 0,Y 142.19,Z 872.804,A -85,B 0,C 180,E1 -25422.142,E2 -25422.142} C_VEL
LIN {X 0,Y 144.177,Z 880.037,A -85,B 0,C 180,E1 -25426.402,E2 -25426.402} C_VEL
LIN {X 0,Y 145.375,Z 887.548,A -85,B 0,C 180,E1 -25430.67,E2 -25430.67} C_VEL
LIN {X 0,Y 145.674,Z 891.703,A -85,B 0,C 180,E1 -25433.05,E2 -25433.05} C_VEL
LIN {X 0,Y 145.315,Z 893.13,A -85,B 0,C 180,E1 -25433.735,E2 -25433.735} C_VEL
LIN {X 0,Y 141.131,Z 900.46,A -85,B 0,C 180,E1 -25436.78,E2 -25436.78} C_VEL
LIN {X 0,Y 136.775,Z 907.825,A -85,B 0,C 180,E1 -25440.871,E2 -25440.871} C_VEL
LIN {X 0,Y 133.137,Z 913.503,A -85,B 0,C 180,E1 -25445.014,E2 -25445.014} C_VEL
LIN {X 0,Y 129.626,Z 918.138,A -85,B 0,C 180,E1 -25449.359,E2 -25449.359} C_VEL
LIN {X 0,Y 126.918,Z 921.658,A -85,B 0,C 180,E1 -25453.921,E2 -25453.921} C_VEL
LIN {X 0,Y 125.696,Z 923.444,A -85,B 0,C 180,E1 -25457.071,E2 -25457.071} C_VEL
LIN {X 0,Y 124.742,Z 924.786,A -85,B 0,C 180,E1 -25460.263,E2 -25460.263} C_VEL
LIN {X 0,Y 123.408,Z 926.363,A -85,B 0,C 180,E1 -25466.729,E2 -25466.729} C_VEL
LIN {X 0,Y 123.274,Z 926.583,A -85,B 0,C 180,E1 -25469.994,E2 -25469.994} C_VEL
LIN {X 0,Y 123.921,Z 925.812,A -85,B 0,C 180,E1 -25476.507,E2 -25476.507} C_VEL
LIN {X 0,Y 124.72,Z 924.861,A -85,B 0,C 180,E1 -25479.727,E2 -25479.727} C_VEL
LIN {X 0,Y 125.671,Z 923.551,A -85,B 0,C 180,E1 -25482.92,E2 -25482.92} C_VEL
LIN {X 0,Y 127.7,Z 920.763,A -85,B 0,C 180,E1 -25487.613,E2 -25487.613} C_VEL
LIN {X 0,Y 130.762,Z 916.911,A -85,B 0,C 180,E1 -25492.094,E2 -25492.094} C_VEL
LIN {X 0,Y 134.274,Z 911.978,A -85,B 0,C 180,E1 -25496.41,E2 -25496.41} C_VEL
LIN {X 0,Y 138.165,Z 905.788,A -85,B 0,C 180,E1 -25500.569,E2 -25500.569} C_VEL
LIN {X 0,Y 141.827,Z 899.474,A -85,B 0,C 180,E1 -25503.875,E2 -25503.875} C_VEL
LIN {X 0,Y 145.214,Z 893.514,A -85,B 0,C 180,E1 -25506.303,E2 -25506.303} C_VEL
LIN {X 0,Y 145.759,Z 892.045,A -85,B 0,C 180,E1 -25506.955,E2 -25506.955} C_VEL
LIN {X 0,Y 145.293,Z 886.451,A -85,B 0,C 180,E1 -25510.169,E2 -25510.169} C_VEL
LIN {X 0,Y 143.897,Z 878.393,A -85,B 0,C 180,E1 -25514.746,E2 -25514.746} C_VEL
LIN {X 0,Y 141.974,Z 871.637,A -85,B 0,C 180,E1 -25518.728,E2 -25518.728} C_VEL
LIN {X 0,Y 139.575,Z 865.18,A -85,B 0,C 180,E1 -25522.826,E2 -25522.826} C_VEL
LIN {X 0,Y 136.568,Z 858.999,A -85,B 0,C 180,E1 -25527.293,E2 -25527.293} C_VEL
LIN {X 0,Y 133.629,Z 853.694,A -85,B 0,C 180,E1 -25531.748,E2 -25531.748} C_VEL
LIN {X 0,Y 129.954,Z 848.111,A -85,B 0,C 180,E1 -25537.755,E2 -25537.755} C_VEL
LIN {X 0,Y 127.755,Z 845.33,A -85,B 0,C 180,E1 -25541.974,E2 -25541.974} C_VEL
LIN {X 0,Y 127.121,Z 843.159,A -85,B 0,C 180,E1 -25543.953,E2 -25543.953} C_VEL
LIN {X 0,Y 123.859,Z 839.955,A -85,B 0,C 180,E1 -25559.187,E2 -25559.187} C_VEL
LIN {X 0,Y 123.93,Z 840.052,A -85,B 0,C 180,E1 -25560.812,E2 -25560.812} C_VEL
LIN {X 0,Y 124.334,Z 841.792,A -85,B 0,C 180,E1 -25565.067,E2 -25565.067} C_VEL
LIN {X 0,Y 125.87,Z 845.359,A -85,B 0,C 180,E1 -25571.066,E2 -25571.066} C_VEL
LIN {X 0,Y 128.595,Z 849.723,A -85,B 0,C 180,E1 -25576.878,E2 -25576.878} C_VEL
LIN {X 0,Y 130.51,Z 854.526,A -85,B 0,C 180,E1 -25580.489,E2 -25580.489} C_VEL
LIN {X 0,Y 132.856,Z 858.092,A -85,B 0,C 180,E1 -25583.685,E2 -25583.685} C_VEL
LIN {X 0,Y 134.851,Z 863.048,A -85,B 0,C 180,E1 -25586.608,E2 -25586.608} C_VEL
LIN {X 0,Y 135.847,Z 864.663,A -85,B 0,C 180,E1 -25587.75,E2 -25587.75} C_VEL
LIN {X 0,Y 137.344,Z 868.968,A -85,B 0,C 180,E1 -25589.885,E2 -25589.885} C_VEL
LIN {X 0,Y 138.528,Z 871.734,A -85,B 0,C 180,E1 -25591.333,E2 -25591.333} C_VEL
LIN {X 0,Y 140.804,Z 878.674,A -85,B 0,C 180,E1 -25594.459,E2 -25594.459} C_VEL
LIN {X 0,Y 143.123,Z 886.768,A -85,B 0,C 180,E1 -25597.867,E2 -25597.867} C_VEL
LIN {X 0,Y 143.71,Z 889.846,A -85,B 0,C 180,E1 -25599.023,E2 -25599.023} C_VEL
LIN {X 0,Y 142.351,Z 901.406,A -85,B 0,C 180,E1 -25602.229,E2 -25602.229} C_VEL
LIN {X 0,Y 140.329,Z 911.832,A -85,B 0,C 180,E1 -25605.488,E2 -25605.488} C_VEL
LIN {X 0,Y 137.522,Z 922.122,A -85,B 0,C 180,E1 -25609.221,E2 -25609.221} C_VEL
LIN {X 0,Y 134.507,Z 930.989,A -85,B 0,C 180,E1 -25613.075,E2 -25613.075} C_VEL
LIN {X 0,Y 130.97,Z 939.414,A -85,B 0,C 180,E1 -25617.554,E2 -25617.554} C_VEL
LIN {X 0,Y 128.665,Z 944.036,A -85,B 0,C 180,E1 -25620.561,E2 -25620.561} C_VEL
LIN {X 0,Y 125.253,Z 949.76,A -85,B 0,C 180,E1 -25625.12,E2 -25625.12} C_VEL
LIN {X 0,Y 122.847,Z 954.326,A -85,B 0,C 180,E1 -25629.931,E2 -25629.931} C_VEL
LIN {X 0,Y 121.476,Z 957.848,A -85,B 0,C 180,E1 -25634.916,E2 -25634.916} C_VEL
LIN {X 0,Y 121.042,Z 960.698,A -85,B 0,C 180,E1 -25640.773,E2 -25640.773} C_VEL
LIN {X 0,Y 121.596,Z 962.296,A -85,B 0,C 180,E1 -25646.693,E2 -25646.693} C_VEL
LIN {X 0,Y 122.128,Z 962.61,A -85,B 0,C 180,E1 -25650.006,E2 -25650.006} C_VEL
LIN {X 0,Y 121.607,Z 962.28,A -85,B 0,C 180,E1 -25653.319,E2 -25653.319} C_VEL
LIN {X 0,Y 121.127,Z 960.577,A -85,B 0,C 180,E1 -25659.471,E2 -25659.471} C_VEL
LIN {X 0,Y 121.749,Z 957.824,A -85,B 0,C 180,E1 -25665.062,E2 -25665.062} C_VEL
LIN {X 0,Y 123.496,Z 954.34,A -85,B 0,C 180,E1 -25669.971,E2 -25669.971} C_VEL
LIN {X 0,Y 126.318,Z 949.819,A -85,B 0,C 180,E1 -25674.669,E2 -25674.669} C_VEL
LIN {X 0,Y 128.021,Z 947.549,A -85,B 0,C 180,E1 -25676.716,E2 -25676.716} C_VEL
LIN {X 0,Y 132.431,Z 947.692,A -85,B 0,C 180,E1 -25682.058,E2 -25682.058} C_VEL
LIN {X 0,Y 138.83,Z 946.973,A -85,B 0,C 180,E1 -25687.413,E2 -25687.413} C_VEL
LIN {X 0,Y 146.259,Z 945.415,A -85,B 0,C 180,E1 -25692.283,E2 -25692.283} C_VEL
LIN {X 0,Y 154.932,Z 943.126,A -85,B 0,C 180,E1 -25696.54,E2 -25696.54} C_VEL
LIN {X 0,Y 161.762,Z 940.975,A -85,B 0,C 180,E1 -25699.33,E2 -25699.33} C_VEL
LIN {X 0,Y 164.225,Z 940.006,A -85,B 0,C 180,E1 -25700.387,E2 -25700.387} C_VEL
LIN {X 0,Y 165.167,Z 939.322,A -85,B 0,C 180,E1 -25701.362,E2 -25701.362} C_VEL
LIN {X 0,Y 156.985,Z 938.642,A -85,B 0,C 180,E1 -25704.409,E2 -25704.409} C_VEL
LIN {X 0,Y 148.112,Z 936.635,A -85,B 0,C 180,E1 -25708.536,E2 -25708.536} C_VEL
LIN {X 0,Y 138.494,Z 932.41,A -85,B 0,C 180,E1 -25714.447,E2 -25714.447} C_VEL
LIN {X 0,Y 132.225,Z 927.572,A -85,B 0,C 180,E1 -25719.789,E2 -25719.789} C_VEL
LIN {X 0,Y 130.906,Z 926.167,A -85,B 0,C 180,E1 -25721.191,E2 -25721.191} C_VEL
LIN {X 0,Y 128.427,Z 923.893,A -85,B 0,C 180,E1 -25723.324,E2 -25723.324} C_VEL
LIN {X 0,Y 123.252,Z 919.528,A -85,B 0,C 180,E1 -25726.627,E2 -25726.627} C_VEL
LIN {X 0,Y 118.605,Z 914.532,A -85,B 0,C 180,E1 -25730.063,E2 -25730.063} C_VEL
LIN {X 0,Y 117.036,Z 911.232,A -85,B 0,C 180,E1 -25732.352,E2 -25732.352} C_VEL
LIN {X 0,Y 115.446,Z 902.634,A -85,B 0,C 180,E1 -25738.256,E2 -25738.256} C_VEL
LIN {X 0,Y 115.127,Z 893.577,A -85,B 0,C 180,E1 -25743.5,E2 -25743.5} C_VEL
LIN {X 0,Y 115.72,Z 883.095,A -85,B 0,C 180,E1 -25748.733,E2 -25748.733} C_VEL
LIN {X 0,Y 116.912,Z 869.009,A -85,B 0,C 180,E1 -25754.397,E2 -25754.397} C_VEL
LIN {X 0,Y 116.93,Z 868.64,A -85,B 0,C 180,E1 -25754.637,E2 -25754.637} C_VEL
LIN {X 0,Y 117.21,Z 869.013,A -85,B 0,C 180,E1 -25755.813,E2 -25755.813} C_VEL
LIN {X 0,Y 118.299,Z 868.168,A -85,B 0,C 180,E1 -25757.28,E2 -25757.28} C_VEL
LIN {X 0,Y 121.026,Z 864.963,A -85,B 0,C 180,E1 -25759.506,E2 -25759.506} C_VEL
LIN {X 0,Y 124.509,Z 860.19,A -85,B 0,C 180,E1 -25761.525,E2 -25761.525} C_VEL
LIN {X 0,Y 125.816,Z 859.738,A -85,B 0,C 180,E1 -25763.018,E2 -25763.018} C_VEL
LIN {X 0,Y 128.981,Z 857.977,A -85,B 0,C 180,E1 -25765.844,E2 -25765.844} C_VEL
LIN {X 0,Y 129.926,Z 859.171,A -85,B 0,C 180,E1 -25767.373,E2 -25767.373} C_VEL
LIN {X 0,Y 132.442,Z 864.392,A -85,B 0,C 180,E1 -25772.049,E2 -25772.049} C_VEL
LIN {X 0,Y 135.292,Z 871.565,A -85,B 0,C 180,E1 -25777.464,E2 -25777.464} C_VEL
LIN {X 0,Y 137.241,Z 877.898,A -85,B 0,C 180,E1 -25781.738,E2 -25781.738} C_VEL
LIN {X 0,Y 138.502,Z 883.409,A -85,B 0,C 180,E1 -25785.268,E2 -25785.268} C_VEL
LIN {X 0,Y 139.403,Z 890.836,A -85,B 0,C 180,E1 -25789.869,E2 -25789.869} C_VEL
LIN {X 0,Y 139.506,Z 894.393,A -85,B 0,C 180,E1 -25792.086,E2 -25792.086} C_VEL
LIN {X 0,Y 134.518,Z 902.81,A -85,B 0,C 180,E1 -25795.825,E2 -25795.825} C_VEL
LIN {X 0,Y 130.688,Z 908.849,A -85,B 0,C 180,E1 -25799.366,E2 -25799.366} C_VEL
LIN {X 0,Y 126.806,Z 914.535,A -85,B 0,C 180,E1 -25803.674,E2 -25803.674} C_VEL
LIN {X 0,Y 123.078,Z 919.17,A -85,B 0,C 180,E1 -25808.207,E2 -25808.207} C_VEL
LIN {X 0,Y 120.184,Z 922.69,A -85,B 0,C 180,E1 -25812.993,E2 -25812.993} C_VEL
LIN {X 0,Y 118.86,Z 924.476,A -85,B 0,C 180,E1 -25816.313,E2 -25816.313} C_VEL
LIN {X 0,Y 117.824,Z 925.818,A -85,B 0,C 180,E1 -25819.686,E2 -25819.686} C_VEL
LIN {X 0,Y 116.396,Z 927.394,A -85,B 0,C 180,E1 -25826.532,E2 -25826.532} C_VEL
LIN {X 0,Y 116.267,Z 927.611,A -85,B 0,C 180,E1 -25829.994,E2 -25829.994} C_VEL
LIN {X 0,Y 116.945,Z 926.843,A -85,B 0,C 180,E1 -25836.897,E2 -25836.897} C_VEL
LIN {X 0,Y 117.803,Z 925.892,A -85,B 0,C 180,E1 -25840.304,E2 -25840.304} C_VEL
LIN {X 0,Y 118.836,Z 924.582,A -85,B 0,C 180,E1 -25843.677,E2 -25843.677} C_VEL
LIN {X 0,Y 121.023,Z 921.793,A -85,B 0,C 180,E1 -25848.62,E2 -25848.62} C_VEL
LIN {X 0,Y 124.281,Z 917.941,A -85,B 0,C 180,E1 -25853.312,E2 -25853.312} C_VEL
LIN {X 0,Y 128.026,Z 913.007,A -85,B 0,C 180,E1 -25857.808,E2 -25857.808} C_VEL
LIN {X 0,Y 132.164,Z 906.817,A -85,B 0,C 180,E1 -25862.118,E2 -25862.118} C_VEL
LIN {X 0,Y 136.051,Z 900.503,A -85,B 0,C 180,E1 -25865.524,E2 -25865.524} C_VEL
LIN {X 0,Y 139.478,Z 894.762,A -85,B 0,C 180,E1 -25867.93,E2 -25867.93} C_VEL
LIN {X 0,Y 139.282,Z 888.802,A -85,B 0,C 180,E1 -25871.622,E2 -25871.622} C_VEL
LIN {X 0,Y 138.246,Z 881.58,A -85,B 0,C 180,E1 -25876.095,E2 -25876.095} C_VEL
LIN {X 0,Y 136.541,Z 874.732,A -85,B 0,C 180,E1 -25880.531,E2 -25880.531} C_VEL
LIN {X 0,Y 134.333,Z 868.662,A -85,B 0,C 180,E1 -25884.865,E2 -25884.865} C_VEL
LIN {X 0,Y 132.648,Z 864.66,A -85,B 0,C 180,E1 -25888.006,E2 -25888.006} C_VEL
LIN {X 0,Y 130.111,Z 859.529,A -85,B 0,C 180,E1 -25892.669,E2 -25892.669} C_VEL
LIN {X 0,Y 127.707,Z 855.385,A -85,B 0,C 180,E1 -25897.342,E2 -25897.342} C_VEL
LIN {X 0,Y 125.529,Z 852.266,A -85,B 0,C 180,E1 -25902.114,E2 -25902.114} C_VEL
LIN {X 0,Y 124.79,Z 849.846,A -85,B 0,C 180,E1 -25904.902,E2 -25904.902} C_VEL
LIN {X 0,Y 122.346,Z 847.22,A -85,B 0,C 180,E1 -25917.531,E2 -25917.531} C_VEL
LIN {X 0,Y 122.516,Z 846.944,A -85,B 0,C 180,E1 -25920.411,E2 -25920.411} C_VEL
LIN {X 0,Y 122.854,Z 848.816,A -85,B 0,C 180,E1 -25924.922,E2 -25924.922} C_VEL
LIN {X 0,Y 124.342,Z 852.573,A -85,B 0,C 180,E1 -25931.203,E2 -25931.203} C_VEL
LIN {X 0,Y 126.231,Z 856.016,A -85,B 0,C 180,E1 -25935.749,E2 -25935.749} C_VEL
LIN {X 0,Y 128.146,Z 861.302,A -85,B 0,C 180,E1 -25940.046,E2 -25940.046} C_VEL
LIN {X 0,Y 129.64,Z 863.581,A -85,B 0,C 180,E1 -25942.301,E2 -25942.301} C_VEL
LIN {X 0,Y 131.293,Z 868.481,A -85,B 0,C 180,E1 -25945.355,E2 -25945.355} C_VEL
LIN {X 0,Y 132.323,Z 870.676,A -85,B 0,C 180,E1 -25946.837,E2 -25946.837} C_VEL
LIN {X 0,Y 134.565,Z 877.592,A -85,B 0,C 180,E1 -25950.567,E2 -25950.567} C_VEL
LIN {X 0,Y 137.021,Z 886.486,A -85,B 0,C 180,E1 -25954.859,E2 -25954.859} C_VEL
LIN {X 0,Y 138.238,Z 892.861,A -85,B 0,C 180,E1 -25957.595,E2 -25957.595} C_VEL
LIN {X 0,Y 136.394,Z 904.182,A -85,B 0,C 180,E1 -25961.017,E2 -25961.017} C_VEL
LIN {X 0,Y 134.012,Z 914.117,A -85,B 0,C 180,E1 -25964.403,E2 -25964.403} C_VEL
LIN {X 0,Y 131.203,Z 923.029,A -85,B 0,C 180,E1 -25967.908,E2 -25967.908} C_VEL
LIN {X 0,Y 127.994,Z 931.467,A -85,B 0,C 180,E1 -25971.858,E2 -25971.858} C_VEL
LIN {X 0,Y 124.256,Z 939.562,A -85,B 0,C 180,E1 -25976.54,E2 -25976.54} C_VEL
LIN {X 0,Y 121.269,Z 944.947,A -85,B 0,C 180,E1 -25980.378,E2 -25980.378} C_VEL
LIN {X 0,Y 117.786,Z 950.373,A -85,B 0,C 180,E1 -25985.319,E2 -25985.319} C_VEL
LIN {X 0,Y 115.497,Z 954.582,A -85,B 0,C 180,E1 -25990.454,E2 -25990.454} C_VEL
LIN {X 0,Y 114.26,Z 957.772,A -85,B 0,C 180,E1 -25995.764,E2 -25995.764} C_VEL
LIN {X 0,Y 113.986,Z 959.787,A -85,B 0,C 180,E1 -26000.578,E2 -26000.578} C_VEL
LIN {X 0,Y 114.517,Z 961.255,A -85,B 0,C 180,E1 -26006.488,E2 -26006.488} C_VEL
LIN {X 0,Y 115.062,Z 961.573,A -85,B 0,C 180,E1 -26010.006,E2 -26010.006} C_VEL
LIN {X 0,Y 114.53,Z 961.239,A -85,B 0,C 180,E1 -26013.524,E2 -26013.524} C_VEL
LIN {X 0,Y 114.076,Z 959.661,A -85,B 0,C 180,E1 -26019.692,E2 -26019.692} C_VEL
LIN {X 0,Y 114.884,Z 956.777,A -85,B 0,C 180,E1 -26025.985,E2 -26025.985} C_VEL
LIN {X 0,Y 116.808,Z 953.29,A -85,B 0,C 180,E1 -26031.168,E2 -26031.168} C_VEL
LIN {X 0,Y 119.917,Z 948.778,A -85,B 0,C 180,E1 -26036.082,E2 -26036.082} C_VEL
LIN {X 0,Y 122.676,Z 945.409,A -85,B 0,C 180,E1 -26039.147,E2 -26039.147} C_VEL
LIN {X 0,Y 129.808,Z 945.62,A -85,B 0,C 180,E1 -26046.559,E2 -26046.559} C_VEL
LIN {X 0,Y 141.136,Z 944.085,A -85,B 0,C 180,E1 -26054.205,E2 -26054.205} C_VEL
LIN {X 0,Y 154.98,Z 940.939,A -85,B 0,C 180,E1 -26060.442,E2 -26060.442} C_VEL
LIN {X 0,Y 156.331,Z 940.563,A -85,B 0,C 180,E1 -26060.995,E2 -26060.995} C_VEL
LIN {X 0,Y 146.621,Z 938.681,A -85,B 0,C 180,E1 -26064.886,E2 -26064.886} C_VEL
LIN {X 0,Y 137.869,Z 935.559,A -85,B 0,C 180,E1 -26069.352,E2 -26069.352} C_VEL
LIN {X 0,Y 130.353,Z 931.312,A -85,B 0,C 180,E1 -26074.449,E2 -26074.449} C_VEL
LIN {X 0,Y 124.198,Z 925.791,A -85,B 0,C 180,E1 -26080.152,E2 -26080.152} C_VEL
LIN {X 0,Y 119.767,Z 918.799,A -85,B 0,C 180,E1 -26086.425,E2 -26086.425} C_VEL
LIN {X 0,Y 117.077,Z 911.392,A -85,B 0,C 180,E1 -26092.238,E2 -26092.238} C_VEL
LIN {X 0,Y 117.036,Z 911.232,A -85,B 0,C 180,E1 -26092.352,E2 -26092.352} C_VEL
LIN {X 0,Y 115.647,Z 907.917,A -85,B 0,C 180,E1 -26094.625,E2 -26094.625} C_VEL
LIN {X 0,Y 112.047,Z 901.761,A -85,B 0,C 180,E1 -26098.133,E2 -26098.133} C_VEL
LIN {X 0,Y 108.868,Z 895.162,A -85,B 0,C 180,E1 -26101.647,E2 -26101.647} C_VEL
LIN {X 0,Y 108.205,Z 890.956,A -85,B 0,C 180,E1 -26103.837,E2 -26103.837} C_VEL
LIN {X 0,Y 108.788,Z 881.063,A -85,B 0,C 180,E1 -26108.826,E2 -26108.826} C_VEL
LIN {X 0,Y 108.695,Z 881.312,A -85,B 0,C 180,E1 -26109.303,E2 -26109.303} C_VEL
LIN {X 0,Y 109.175,Z 881.027,A -85,B 0,C 180,E1 -26111.135,E2 -26111.135} C_VEL
LIN {X 0,Y 110.35,Z 879.772,A -85,B 0,C 180,E1 -26112.88,E2 -26112.88} C_VEL
LIN {X 0,Y 112.897,Z 876.742,A -85,B 0,C 180,E1 -26115.342,E2 -26115.342} C_VEL
LIN {X 0,Y 113.939,Z 875.424,A -85,B 0,C 180,E1 -26116.115,E2 -26116.115} C_VEL
LIN {X 0,Y 115.082,Z 874.683,A -85,B 0,C 180,E1 -26117.779,E2 -26117.779} C_VEL
LIN {X 0,Y 116.54,Z 873.522,A -85,B 0,C 180,E1 -26119.371,E2 -26119.371} C_VEL
LIN {X 0,Y 119.535,Z 870.463,A -85,B 0,C 180,E1 -26121.561,E2 -26121.561} C_VEL
LIN {X 0,Y 123.132,Z 866.258,A -85,B 0,C 180,E1 -26123.55,E2 -26123.55} C_VEL
LIN {X 0,Y 126.229,Z 864.942,A -85,B 0,C 180,E1 -26126.45,E2 -26126.45} C_VEL
LIN {X 0,Y 128.477,Z 870.499,A -85,B 0,C 180,E1 -26131.753,E2 -26131.753} C_VEL
LIN {X 0,Y 130.423,Z 876.092,A -85,B 0,C 180,E1 -26136.353,E2 -26136.353} C_VEL
LIN {X 0,Y 131.958,Z 882.089,A -85,B 0,C 180,E1 -26140.799,E2 -26140.799} C_VEL
LIN {X 0,Y 133.024,Z 888.318,A -85,B 0,C 180,E1 -26145.126,E2 -26145.126} C_VEL
LIN {X 0,Y 133.422,Z 895.312,A -85,B 0,C 180,E1 -26149.86,E2 -26149.86} C_VEL
LIN {X 0,Y 133.353,Z 896.664,A -85,B 0,C 180,E1 -26150.764,E2 -26150.764} C_VEL
LIN {X 0,Y 128.775,Z 903.842,A -85,B 0,C 180,E1 -26154.071,E2 -26154.071} C_VEL
LIN {X 0,Y 124.197,Z 910.6,A -85,B 0,C 180,E1 -26158.208,E2 -26158.208} C_VEL
LIN {X 0,Y 120.552,Z 915.568,A -85,B 0,C 180,E1 -26162.194,E2 -26162.194} C_VEL
LIN {X 0,Y 116.586,Z 920.202,A -85,B 0,C 180,E1 -26166.925,E2 -26166.925} C_VEL
LIN {X 0,Y 113.485,Z 923.722,A -85,B 0,C 180,E1 -26171.956,E2 -26171.956} C_VEL
LIN {X 0,Y 112.046,Z 925.508,A -85,B 0,C 180,E1 -26175.463,E2 -26175.463} C_VEL
LIN {X 0,Y 110.92,Z 926.85,A -85,B 0,C 180,E1 -26179.036,E2 -26179.036} C_VEL
LIN {X 0,Y 109.386,Z 928.425,A -85,B 0,C 180,E1 -26186.31,E2 -26186.31} C_VEL
LIN {X 0,Y 109.258,Z 928.64,A -85,B 0,C 180,E1 -26189.993,E2 -26189.993} C_VEL
LIN {X 0,Y 109.975,Z 927.874,A -85,B 0,C 180,E1 -26197.336,E2 -26197.336} C_VEL
LIN {X 0,Y 110.899,Z 926.923,A -85,B 0,C 180,E1 -26200.953,E2 -26200.953} C_VEL
LIN {X 0,Y 112.024,Z 925.612,A -85,B 0,C 180,E1 -26204.527,E2 -26204.527} C_VEL
LIN {X 0,Y 114.388,Z 922.824,A -85,B 0,C 180,E1 -26209.743,E2 -26209.743} C_VEL
LIN {X 0,Y 117.863,Z 918.971,A -85,B 0,C 180,E1 -26214.664,E2 -26214.664} C_VEL
LIN {X 0,Y 121.861,Z 914.036,A -85,B 0,C 180,E1 -26219.347,E2 -26219.347} C_VEL
LIN {X 0,Y 126.272,Z 907.846,A -85,B 0,C 180,E1 -26223.812,E2 -26223.812} C_VEL
LIN {X 0,Y 130.398,Z 901.532,A -85,B 0,C 180,E1 -26227.317,E2 -26227.317} C_VEL
LIN {X 0,Y 133.264,Z 897.071,A -85,B 0,C 180,E1 -26229.253,E2 -26229.253} C_VEL
LIN {X 0,Y 133.506,Z 894.162,A -85,B 0,C 180,E1 -26231.147,E2 -26231.147} C_VEL
LIN {X 0,Y 133.033,Z 887.456,A -85,B 0,C 180,E1 -26235.689,E2 -26235.689} C_VEL
LIN {X 0,Y 131.873,Z 880.897,A -85,B 0,C 180,E1 -26240.243,E2 -26240.243} C_VEL
LIN {X 0,Y 130.341,Z 875.265,A -85,B 0,C 180,E1 -26244.479,E2 -26244.479} C_VEL
LIN {X 0,Y 128.876,Z 871.062,A -85,B 0,C 180,E1 -26247.964,E2 -26247.964} C_VEL
LIN {X 0,Y 126.903,Z 866.462,A -85,B 0,C 180,E1 -26252.373,E2 -26252.373} C_VEL
LIN {X 0,Y 124.408,Z 861.281,A -85,B 0,C 180,E1 -26258.457,E2 -26258.457} C_VEL
LIN {X 0,Y 121.921,Z 856.23,A -85,B 0,C 180,E1 -26266.669,E2 -26266.669} C_VEL
LIN {X 0,Y 120.563,Z 853.957,A -85,B 0,C 180,E1 -26278.33,E2 -26278.33} C_VEL
LIN {X 0,Y 120.725,Z 853.866,A -85,B 0,C 180,E1 -26280.417,E2 -26280.417} C_VEL
LIN {X 0,Y 121.186,Z 856.537,A -85,B 0,C 180,E1 -26286.242,E2 -26286.242} C_VEL
LIN {X 0,Y 123.034,Z 861.029,A -85,B 0,C 180,E1 -26293.208,E2 -26293.208} C_VEL
LIN {X 0,Y 123.572,Z 862.481,A -85,B 0,C 180,E1 -26294.82,E2 -26294.82} C_VEL
LIN {X 0,Y 125.432,Z 867.946,A -85,B 0,C 180,E1 -26299.644,E2 -26299.644} C_VEL
LIN {X 0,Y 126.302,Z 869.468,A -85,B 0,C 180,E1 -26301.204,E2 -26301.204} C_VEL
LIN {X 0,Y 128.506,Z 876.518,A -85,B 0,C 180,E1 -26305.946,E2 -26305.946} C_VEL
LIN {X 0,Y 130.353,Z 883.376,A -85,B 0,C 180,E1 -26309.893,E2 -26309.893} C_VEL
LIN {X 0,Y 132.291,Z 892.415,A -85,B 0,C 180,E1 -26314.506,E2 -26314.506} C_VEL
LIN {X 0,Y 132.786,Z 895.743,A -85,B 0,C 180,E1 -26316.073,E2 -26316.073} C_VEL
LIN {X 0,Y 130.368,Z 907.111,A -85,B 0,C 180,E1 -26319.819,E2 -26319.819} C_VEL
LIN {X 0,Y 127.367,Z 917.213,A -85,B 0,C 180,E1 -26323.604,E2 -26323.604} C_VEL
LIN {X 0,Y 123.875,Z 926.569,A -85,B 0,C 180,E1 -26327.756,E2 -26327.756} C_VEL
LIN {X 0,Y 120.173,Z 934.656,A -85,B 0,C 180,E1 -26332.124,E2 -26332.124} C_VEL
LIN {X 0,Y 116.349,Z 941.927,A -85,B 0,C 180,E1 -26337.076,E2 -26337.076} C_VEL
LIN {X 0,Y 112.456,Z 947.666,A -85,B 0,C 180,E1 -26342.057,E2 -26342.057} C_VEL
LIN {X 0,Y 109.493,Z 952.223,A -85,B 0,C 180,E1 -26347.356,E2 -26347.356} C_VEL
LIN {X 0,Y 107.684,Z 955.743,A -85,B 0,C 180,E1 -26352.928,E2 -26352.928} C_VEL
LIN {X 0,Y 106.931,Z 958.875,A -85,B 0,C 180,E1 -26360.357,E2 -26360.357} C_VEL
LIN {X 0,Y 107.436,Z 960.214,A -85,B 0,C 180,E1 -26366.256,E2 -26366.256} C_VEL
LIN {X 0,Y 107.993,Z 960.535,A -85,B 0,C 180,E1 -26370.007,E2 -26370.007} C_VEL
LIN {X 0,Y 107.451,Z 960.198,A -85,B 0,C 180,E1 -26373.757,E2 -26373.757} C_VEL
LIN {X 0,Y 107.023,Z 958.749,A -85,B 0,C 180,E1 -26379.929,E2 -26379.929} C_VEL
LIN {X 0,Y 108.032,Z 955.727,A -85,B 0,C 180,E1 -26387.029,E2 -26387.029} C_VEL
LIN {X 0,Y 110.186,Z 952.242,A -85,B 0,C 180,E1 -26392.508,E2 -26392.508} C_VEL
LIN {X 0,Y 113.605,Z 947.738,A -85,B 0,C 180,E1 -26397.651,E2 -26397.651} C_VEL
LIN {X 0,Y 117.597,Z 943.102,A -85,B 0,C 180,E1 -26401.787,E2 -26401.787} C_VEL
LIN {X 0,Y 121.364,Z 943.525,A -85,B 0,C 180,E1 -26405.833,E2 -26405.833} C_VEL
LIN {X 0,Y 128.043,Z 943.472,A -85,B 0,C 180,E1 -26411.204,E2 -26411.204} C_VEL
LIN {X 0,Y 140.763,Z 941.869,A -85,B 0,C 180,E1 -26418.504,E2 -26418.504} C_VEL
LIN {X 0,Y 145.56,Z 941.019,A -85,B 0,C 180,E1 -26420.587,E2 -26420.587} C_VEL
LIN {X 0,Y 145.779,Z 940.699,A -85,B 0,C 180,E1 -26421.191,E2 -26421.191} C_VEL
LIN {X 0,Y 136.227,Z 937.668,A -85,B 0,C 180,E1 -26425.424,E2 -26425.424} C_VEL
LIN {X 0,Y 129.76,Z 934.693,A -85,B 0,C 180,E1 -26429.034,E2 -26429.034} C_VEL
LIN {X 0,Y 123.987,Z 931.058,A -85,B 0,C 180,E1 -26433.034,E2 -26433.034} C_VEL
LIN {X 0,Y 117.583,Z 925.024,A -85,B 0,C 180,E1 -26438.984,E2 -26438.984} C_VEL
LIN {X 0,Y 113.929,Z 919.636,A -85,B 0,C 180,E1 -26443.883,E2 -26443.883} C_VEL
LIN {X 0,Y 111.247,Z 913.389,A -85,B 0,C 180,E1 -26449.075,E2 -26449.075} C_VEL
LIN {X 0,Y 108.966,Z 904.779,A -85,B 0,C 180,E1 -26455.376,E2 -26455.376} C_VEL
LIN {X 0,Y 108.293,Z 895.994,A -85,B 0,C 180,E1 -26460.93,E2 -26460.93} C_VEL
LIN {X 0,Y 108.205,Z 890.956,A -85,B 0,C 180,E1 -26463.837,E2 -26463.837} C_VEL
LIN {X 0,Y 108.221,Z 888.481,A -85,B 0,C 180,E1 -26465.411,E2 -26465.411} C_VEL
LIN {X 0,Y 108.282,Z 885.759,A -85,B 0,C 180,E1 -26468.14,E2 -26468.14} C_VEL
LIN {X 0,Y 108.605,Z 883.944,A -85,B 0,C 180,E1 -26471.089,E2 -26471.089} C_VEL
LIN {X 0,Y 110.806,Z 881.451,A -85,B 0,C 180,E1 -26477.165,E2 -26477.165} C_VEL
LIN {X 0,Y 112.161,Z 880.526,A -85,B 0,C 180,E1 -26479.055,E2 -26479.055} C_VEL
LIN {X 0,Y 114.659,Z 878.721,A -85,B 0,C 180,E1 -26481.578,E2 -26481.578} C_VEL
LIN {X 0,Y 118.134,Z 875.568,A -85,B 0,C 180,E1 -26483.843,E2 -26483.843} C_VEL
LIN {X 0,Y 121.649,Z 871.999,A -85,B 0,C 180,E1 -26485.677,E2 -26485.677} C_VEL
LIN {X 0,Y 122.886,Z 872.141,A -85,B 0,C 180,E1 -26487.228,E2 -26487.228} C_VEL
LIN {X 0,Y 124.56,Z 877.093,A -85,B 0,C 180,E1 -26492.175,E2 -26492.175} C_VEL
LIN {X 0,Y 125.742,Z 881.689,A -85,B 0,C 180,E1 -26496.16,E2 -26496.16} C_VEL
LIN {X 0,Y 126.78,Z 887.294,A -85,B 0,C 180,E1 -26500.643,E2 -26500.643} C_VEL
LIN {X 0,Y 127.352,Z 892.965,A -85,B 0,C 180,E1 -26504.925,E2 -26504.925} C_VEL
LIN {X 0,Y 127.389,Z 897.815,A -85,B 0,C 180,E1 -26508.538,E2 -26508.538} C_VEL
LIN {X 0,Y 126.984,Z 899.273,A -85,B 0,C 180,E1 -26509.428,E2 -26509.428} C_VEL
LIN {X 0,Y 121.383,Z 907.381,A -85,B 0,C 180,E1 -26513.59,E2 -26513.59} C_VEL
LIN {X 0,Y 117.305,Z 912.892,A -85,B 0,C 180,E1 -26517.363,E2 -26517.363} C_VEL
LIN {X 0,Y 112.926,Z 918.267,A -85,B 0,C 180,E1 -26522.169,E2 -26522.169} C_VEL
LIN {X 0,Y 108.918,Z 922.527,A -85,B 0,C 180,E1 -26527.216,E2 -26527.216} C_VEL
LIN {X 0,Y 106.827,Z 924.754,A -85,B 0,C 180,E1 -26530.789,E2 -26530.789} C_VEL
LIN {X 0,Y 105.26,Z 926.54,A -85,B 0,C 180,E1 -26534.503,E2 -26534.503} C_VEL
LIN {X 0,Y 104.031,Z 927.881,A -85,B 0,C 180,E1 -26538.3,E2 -26538.3} C_VEL
LIN {X 0,Y 102.377,Z 929.457,A -85,B 0,C 180,E1 -26546.057,E2 -26546.057} C_VEL
LIN {X 0,Y 102.247,Z 929.67,A -85,B 0,C 180,E1 -26549.993,E2 -26549.993} C_VEL
LIN {X 0,Y 102.372,Z 929.487,A -85,B 0,C 180,E1 -26553.929,E2 -26553.929} C_VEL
LIN {X 0,Y 104.012,Z 927.953,A -85,B 0,C 180,E1 -26561.688,E2 -26561.688} C_VEL
LIN {X 0,Y 105.239,Z 926.643,A -85,B 0,C 180,E1 -26565.486,E2 -26565.486} C_VEL
LIN {X 0,Y 107.801,Z 923.854,A -85,B 0,C 180,E1 -26571.005,E2 -26571.005} C_VEL
LIN {X 0,Y 111.517,Z 920.001,A -85,B 0,C 180,E1 -26576.17,E2 -26576.17} C_VEL
LIN {X 0,Y 115.792,Z 915.065,A -85,B 0,C 180,E1 -26581.05,E2 -26581.05} C_VEL
LIN {X 0,Y 121.339,Z 907.679,A -85,B 0,C 180,E1 -26586.411,E2 -26586.411} C_VEL
LIN {X 0,Y 125.905,Z 901.099,A -85,B 0,C 180,E1 -26589.928,E2 -26589.928} C_VEL
LIN {X 0,Y 126.924,Z 899.636,A -85,B 0,C 180,E1 -26590.58,E2 -26590.58} C_VEL
LIN {X 0,Y 127.439,Z 898.189,A -85,B 0,C 180,E1 -26591.427,E2 -26591.427} C_VEL
LIN {X 0,Y 127.421,Z 892.316,A -85,B 0,C 180,E1 -26595.8,E2 -26595.8} C_VEL
LIN {X 0,Y 126.912,Z 887.101,A -85,B 0,C 180,E1 -26599.706,E2 -26599.706} C_VEL
LIN {X 0,Y 126.028,Z 882.193,A -85,B 0,C 180,E1 -26603.615,E2 -26603.615} C_VEL
LIN {X 0,Y 124.875,Z 877.631,A -85,B 0,C 180,E1 -26607.575,E2 -26607.575} C_VEL
LIN {X 0,Y 123.552,Z 873.553,A -85,B 0,C 180,E1 -26611.557,E2 -26611.557} C_VEL
LIN {X 0,Y 121.916,Z 869.65,A -85,B 0,C 180,E1 -26616.201,E2 -26616.201} C_VEL
LIN {X 0,Y 120.915,Z 867.107,A -85,B 0,C 180,E1 -26619.589,E2 -26619.589} C_VEL
LIN {X 0,Y 119.365,Z 863.175,A -85,B 0,C 180,E1 -26626.378,E2 -26626.378} C_VEL
LIN {X 0,Y 118.291,Z 861.529,A -85,B 0,C 180,E1 -26633.175,E2 -26633.175} C_VEL
LIN {X 0,Y 118.553,Z 860.569,A -85,B 0,C 180,E1 -26640,E2 -26640} C_VEL
LIN {X 0,Y 119.006,Z 863.734,A -85,B 0,C 180,E1 -26646.783,E2 -26646.783} C_VEL
LIN {X 0,Y 120.083,Z 866.947,A -85,B 0,C 180,E1 -26651.82,E2 -26651.82} C_VEL
LIN {X 0,Y 120.538,Z 868.289,A -85,B 0,C 180,E1 -26653.487,E2 -26653.487} C_VEL
LIN {X 0,Y 121.99,Z 873.614,A -85,B 0,C 180,E1 -26658.473,E2 -26658.473} C_VEL
LIN {X 0,Y 122.706,Z 875.193,A -85,B 0,C 180,E1 -26660.099,E2 -26660.099} C_VEL
LIN {X 0,Y 124.596,Z 882.891,A -85,B 0,C 180,E1 -26665.527,E2 -26665.527} C_VEL
LIN {X 0,Y 125.903,Z 888.926,A -85,B 0,C 180,E1 -26669.237,E2 -26669.237} C_VEL
LIN {X 0,Y 127.274,Z 897.847,A -85,B 0,C 180,E1 -26674.088,E2 -26674.088} C_VEL
LIN {X 0,Y 126.669,Z 901.322,A -85,B 0,C 180,E1 -26675.399,E2 -26675.399} C_VEL
LIN {X 0,Y 123.521,Z 912.426,A -85,B 0,C 180,E1 -26679.507,E2 -26679.507} C_VEL
LIN {X 0,Y 120.307,Z 920.925,A -85,B 0,C 180,E1 -26683.105,E2 -26683.105} C_VEL
LIN {X 0,Y 116.517,Z 929.507,A -85,B 0,C 180,E1 -26687.451,E2 -26687.451} C_VEL
LIN {X 0,Y 112.312,Z 937.412,A -85,B 0,C 180,E1 -26692.411,E2 -26692.411} C_VEL
LIN {X 0,Y 109,Z 942.862,A -85,B 0,C 180,E1 -26696.662,E2 -26696.662} C_VEL
LIN {X 0,Y 104.943,Z 948.273,A -85,B 0,C 180,E1 -26702.053,E2 -26702.053} C_VEL
LIN {X 0,Y 102.091,Z 952.478,A -85,B 0,C 180,E1 -26707.76,E2 -26707.76} C_VEL
LIN {X 0,Y 100.425,Z 955.668,A -85,B 0,C 180,E1 -26713.752,E2 -26713.752} C_VEL
LIN {X 0,Y 99.887,Z 957.951,A -85,B 0,C 180,E1 -26720.076,E2 -26720.076} C_VEL
LIN {X 0,Y 100.351,Z 959.171,A -85,B 0,C 180,E1 -26725.991,E2 -26725.991} C_VEL
LIN {X 0,Y 100.921,Z 959.497,A -85,B 0,C 180,E1 -26730.007,E2 -26730.007} C_VEL
LIN {X 0,Y 100.372,Z 959.156,A -85,B 0,C 180,E1 -26734.022,E2 -26734.022} C_VEL
LIN {X 0,Y 100.085,Z 957.213,A -85,B 0,C 180,E1 -26742.168,E2 -26742.168} C_VEL
LIN {X 0,Y 101.242,Z 954.681,A -85,B 0,C 180,E1 -26748.21,E2 -26748.21} C_VEL
LIN {X 0,Y 103.64,Z 951.195,A -85,B 0,C 180,E1 -26754.016,E2 -26754.016} C_VEL
LIN {X 0,Y 107.386,Z 946.698,A -85,B 0,C 180,E1 -26759.403,E2 -26759.403} C_VEL
LIN {X 0,Y 112.838,Z 940.777,A -85,B 0,C 180,E1 -26764.642,E2 -26764.642} C_VEL
LIN {X 0,Y 119.085,Z 941.406,A -85,B 0,C 180,E1 -26770.487,E2 -26770.487} C_VEL
LIN {X 0,Y 127.078,Z 941.205,A -85,B 0,C 180,E1 -26775.976,E2 -26775.976} C_VEL
LIN {X 0,Y 136.246,Z 940.244,A -85,B 0,C 180,E1 -26780.699,E2 -26780.699} C_VEL
LIN {X 0,Y 135.271,Z 939.739,A -85,B 0,C 180,E1 -26781.431,E2 -26781.431} C_VEL
LIN {X 0,Y 128.115,Z 936.883,A -85,B 0,C 180,E1 -26784.83,E2 -26784.83} C_VEL
LIN {X 0,Y 119.636,Z 931.993,A -85,B 0,C 180,E1 -26790.044,E2 -26790.044} C_VEL
LIN {X 0,Y 114.167,Z 927.544,A -85,B 0,C 180,E1 -26794.475,E2 -26794.475} C_VEL
LIN {X 0,Y 108.384,Z 920.384,A -85,B 0,C 180,E1 -26801.082,E2 -26801.082} C_VEL
LIN {X 0,Y 105.266,Z 914.085,A -85,B 0,C 180,E1 -26806.487,E2 -26806.487} C_VEL
LIN {X 0,Y 102.577,Z 905.491,A -85,B 0,C 180,E1 -26813.114,E2 -26813.114} C_VEL
LIN {X 0,Y 101.448,Z 895.121,A -85,B 0,C 180,E1 -26820,E2 -26820} C_VEL
LIN {X 0,Y 101.279,Z 892.553,A -85,B 0,C 180,E1 -26821.74,E2 -26821.74} C_VEL
LIN {X 0,Y 101.198,Z 892.343,A -85,B 0,C 180,E1 -26823.982,E2 -26823.982} C_VEL
LIN {X 0,Y 101.847,Z 891.362,A -85,B 0,C 180,E1 -26825.941,E2 -26825.941} C_VEL
LIN {X 0,Y 102.983,Z 889.863,A -85,B 0,C 180,E1 -26827.845,E2 -26827.845} C_VEL
LIN {X 0,Y 104.456,Z 887.96,A -85,B 0,C 180,E1 -26829.684,E2 -26829.684} C_VEL
LIN {X 0,Y 106.383,Z 886.138,A -85,B 0,C 180,E1 -26833.369,E2 -26833.369} C_VEL
LIN {X 0,Y 107.775,Z 884.819,A -85,B 0,C 180,E1 -26835.12,E2 -26835.12} C_VEL
LIN {X 0,Y 111.586,Z 880.917,A -85,B 0,C 180,E1 -26838.356,E2 -26838.356} C_VEL
LIN {X 0,Y 112.161,Z 880.526,A -85,B 0,C 180,E1 -26839.055,E2 -26839.055} C_VEL
LIN {X 0,Y 115.429,Z 878.777,A -85,B 0,C 180,E1 -26842.826,E2 -26842.826} C_VEL
LIN {X 0,Y 117.435,Z 878.382,A -85,B 0,C 180,E1 -26845.322,E2 -26845.322} C_VEL
LIN {X 0,Y 118.927,Z 879.052,A -85,B 0,C 180,E1 -26847.787,E2 -26847.787} C_VEL
LIN {X 0,Y 119.338,Z 879.918,A -85,B 0,C 180,E1 -26848.981,E2 -26848.981} C_VEL
LIN {X 0,Y 120.351,Z 884.314,A -85,B 0,C 180,E1 -26853.445,E2 -26853.445} C_VEL
LIN {X 0,Y 121.223,Z 890.018,A -85,B 0,C 180,E1 -26858.554,E2 -26858.554} C_VEL
LIN {X 0,Y 121.582,Z 894.698,A -85,B 0,C 180,E1 -26862.541,E2 -26862.541} C_VEL
LIN {X 0,Y 121.387,Z 900.376,A -85,B 0,C 180,E1 -26867.126,E2 -26867.126} C_VEL
LIN {X 0,Y 120.657,Z 901.771,A -85,B 0,C 180,E1 -26867.937,E2 -26867.937} C_VEL
LIN {X 0,Y 114.899,Z 909.611,A -85,B 0,C 180,E1 -26872.282,E2 -26872.282} C_VEL
LIN {X 0,Y 109.865,Z 915.87,A -85,B 0,C 180,E1 -26877.054,E2 -26877.054} C_VEL
LIN {X 0,Y 105.278,Z 920.863,A -85,B 0,C 180,E1 -26882.134,E2 -26882.134} C_VEL
LIN {X 0,Y 101.3,Z 924.753,A -85,B 0,C 180,E1 -26887.561,E2 -26887.561} C_VEL
LIN {X 0,Y 98.508,Z 927.572,A -85,B 0,C 180,E1 -26893.411,E2 -26893.411} C_VEL
LIN {X 0,Y 97.162,Z 928.913,A -85,B 0,C 180,E1 -26897.46,E2 -26897.46} C_VEL
LIN {X 0,Y 95.37,Z 930.488,A -85,B 0,C 180,E1 -26905.766,E2 -26905.766} C_VEL
LIN {X 0,Y 95.234,Z 930.699,A -85,B 0,C 180,E1 -26909.992,E2 -26909.992} C_VEL
LIN {X 0,Y 95.365,Z 930.518,A -85,B 0,C 180,E1 -26914.219,E2 -26914.219} C_VEL
LIN {X 0,Y 97.143,Z 928.984,A -85,B 0,C 180,E1 -26922.527,E2 -26922.527} C_VEL
LIN {X 0,Y 98.487,Z 927.673,A -85,B 0,C 180,E1 -26926.577,E2 -26926.577} C_VEL
LIN {X 0,Y 101.274,Z 924.885,A -85,B 0,C 180,E1 -26932.429,E2 -26932.429} C_VEL
LIN {X 0,Y 105.258,Z 921.031,A -85,B 0,C 180,E1 -26937.857,E2 -26937.857} C_VEL
LIN {X 0,Y 109.836,Z 916.095,A -85,B 0,C 180,E1 -26942.94,E2 -26942.94} C_VEL
LIN {X 0,Y 115.76,Z 908.709,A -85,B 0,C 180,E1 -26948.475,E2 -26948.475} C_VEL
LIN {X 0,Y 120.608,Z 902.126,A -85,B 0,C 180,E1 -26952.068,E2 -26952.068} C_VEL
LIN {X 0,Y 121.453,Z 900.709,A -85,B 0,C 180,E1 -26952.829,E2 -26952.829} C_VEL
LIN {X 0,Y 121.681,Z 895.054,A -85,B 0,C 180,E1 -26957.417,E2 -26957.417} C_VEL
LIN {X 0,Y 121.279,Z 888.986,A -85,B 0,C 180,E1 -26962.523,E2 -26962.523} C_VEL
LIN {X 0,Y 120.229,Z 882.814,A -85,B 0,C 180,E1 -26968.258,E2 -26968.258} C_VEL
LIN {X 0,Y 119.337,Z 879.24,A -85,B 0,C 180,E1 -26972.038,E2 -26972.038} C_VEL
LIN {X 0,Y 118.017,Z 875.267,A -85,B 0,C 180,E1 -26977.131,E2 -26977.131} C_VEL
LIN {X 0,Y 117.232,Z 872.834,A -85,B 0,C 180,E1 -26980.748,E2 -26980.748} C_VEL
LIN {X 0,Y 116.359,Z 869.986,A -85,B 0,C 180,E1 -26986.019,E2 -26986.019} C_VEL
LIN {X 0,Y 115.921,Z 868.786,A -85,B 0,C 180,E1 -26989.52,E2 -26989.52} C_VEL
LIN {X 0,Y 115.626,Z 867.61,A -85,B 0,C 180,E1 -26996.515,E2 -26996.515} C_VEL
LIN {X 0,Y 115.984,Z 867.33,A -85,B 0,C 180,E1 -27000,E2 -27000} C_VEL
LIN {X 0,Y 116.012,Z 868.787,A -85,B 0,C 180,E1 -27003.473,E2 -27003.473} C_VEL
LIN {X 0,Y 116.882,Z 872.725,A -85,B 0,C 180,E1 -27010.392,E2 -27010.392} C_VEL
LIN {X 0,Y 117.244,Z 873.985,A -85,B 0,C 180,E1 -27012.111,E2 -27012.111} C_VEL
LIN {X 0,Y 118.86,Z 880.681,A -85,B 0,C 180,E1 -27018.926,E2 -27018.926} C_VEL
LIN {X 0,Y 119.966,Z 886.289,A -85,B 0,C 180,E1 -27023.293,E2 -27023.293} C_VEL
LIN {X 0,Y 120.973,Z 892.879,A -85,B 0,C 180,E1 -27027.695,E2 -27027.695} C_VEL
LIN {X 0,Y 121.731,Z 900.204,A -85,B 0,C 180,E1 -27032.078,E2 -27032.078} C_VEL
LIN {X 0,Y 121.724,Z 901.718,A -85,B 0,C 180,E1 -27032.859,E2 -27032.859} C_VEL
LIN {X 0,Y 118.477,Z 911.847,A -85,B 0,C 180,E1 -27036.822,E2 -27036.822} C_VEL
LIN {X 0,Y 115.253,Z 919.814,A -85,B 0,C 180,E1 -27040.349,E2 -27040.349} C_VEL
LIN {X 0,Y 111.394,Z 927.889,A -85,B 0,C 180,E1 -27044.549,E2 -27044.549} C_VEL
LIN {X 0,Y 107.326,Z 935.106,A -85,B 0,C 180,E1 -27049.103,E2 -27049.103} C_VEL
LIN {X 0,Y 102.989,Z 941.91,A -85,B 0,C 180,E1 -27054.558,E2 -27054.558} C_VEL
LIN {X 0,Y 98.684,Z 947.224,A -85,B 0,C 180,E1 -27060.107,E2 -27060.107} C_VEL
LIN {X 0,Y 95.498,Z 951.427,A -85,B 0,C 180,E1 -27066.132,E2 -27066.132} C_VEL
LIN {X 0,Y 93.545,Z 954.614,A -85,B 0,C 180,E1 -27072.52,E2 -27072.52} C_VEL
LIN {X 0,Y 92.856,Z 957.002,A -85,B 0,C 180,E1 -27079.715,E2 -27079.715} C_VEL
LIN {X 0,Y 93.246,Z 958.126,A -85,B 0,C 180,E1 -27085.685,E2 -27085.685} C_VEL
LIN {X 0,Y 93.845,Z 958.458,A -85,B 0,C 180,E1 -27090.008,E2 -27090.008} C_VEL
LIN {X 0,Y 93.272,Z 958.111,A -85,B 0,C 180,E1 -27094.329,E2 -27094.329} C_VEL
LIN {X 0,Y 93.127,Z 956.166,A -85,B 0,C 180,E1 -27103.093,E2 -27103.093} C_VEL
LIN {X 0,Y 94.514,Z 953.636,A -85,B 0,C 180,E1 -27109.557,E2 -27109.557} C_VEL
LIN {X 0,Y 97.182,Z 950.149,A -85,B 0,C 180,E1 -27115.723,E2 -27115.723} C_VEL
LIN {X 0,Y 101.283,Z 945.658,A -85,B 0,C 180,E1 -27121.368,E2 -27121.368} C_VEL
LIN {X 0,Y 106.639,Z 940.04,A -85,B 0,C 180,E1 -27126.388,E2 -27126.388} C_VEL
LIN {X 0,Y 108.424,Z 938.398,A -85,B 0,C 180,E1 -27127.723,E2 -27127.723} C_VEL
LIN {X 0,Y 118.067,Z 939.182,A -85,B 0,C 180,E1 -27135.594,E2 -27135.594} C_VEL
LIN {X 0,Y 124.532,Z 938.958,A -85,B 0,C 180,E1 -27139.479,E2 -27139.479} C_VEL
LIN {X 0,Y 126.062,Z 938.464,A -85,B 0,C 180,E1 -27141.131,E2 -27141.131} C_VEL
LIN {X 0,Y 117.798,Z 934.25,A -85,B 0,C 180,E1 -27145.474,E2 -27145.474} C_VEL
LIN {X 0,Y 109.637,Z 928.286,A -85,B 0,C 180,E1 -27151.265,E2 -27151.265} C_VEL
LIN {X 0,Y 104.569,Z 922.998,A -85,B 0,C 180,E1 -27156.218,E2 -27156.218} C_VEL
LIN {X 0,Y 100.007,Z 915.8,A -85,B 0,C 180,E1 -27162.623,E2 -27162.623} C_VEL
LIN {X 0,Y 96.77,Z 907.401,A -85,B 0,C 180,E1 -27169.539,E2 -27169.539} C_VEL
LIN {X 0,Y 95.501,Z 902.808,A -85,B 0,C 180,E1 -27173.132,E2 -27173.132} C_VEL
LIN {X 0,Y 94.89,Z 902.374,A -85,B 0,C 180,E1 -27175.753,E2 -27175.753} C_VEL
LIN {X 0,Y 95.032,Z 901.468,A -85,B 0,C 180,E1 -27177.881,E2 -27177.881} C_VEL
LIN {X 0,Y 96.474,Z 898.682,A -85,B 0,C 180,E1 -27182.088,E2 -27182.088} C_VEL
LIN {X 0,Y 98.286,Z 896.077,A -85,B 0,C 180,E1 -27188.222,E2 -27188.222} C_VEL
LIN {X 0,Y 101.181,Z 892.935,A -85,B 0,C 180,E1 -27192.028,E2 -27192.028} C_VEL
LIN {X 0,Y 103.519,Z 891.005,A -85,B 0,C 180,E1 -27195.758,E2 -27195.758} C_VEL
LIN {X 0,Y 106.07,Z 888.81,A -85,B 0,C 180,E1 -27198.315,E2 -27198.315} C_VEL
LIN {X 0,Y 109.201,Z 886.084,A -85,B 0,C 180,E1 -27200.742,E2 -27200.742} C_VEL
LIN {X 0,Y 112.709,Z 883.711,A -85,B 0,C 180,E1 -27203.911,E2 -27203.911} C_VEL
LIN {X 0,Y 116.885,Z 880.288,A -85,B 0,C 180,E1 -27206.346,E2 -27206.346} C_VEL
LIN {X 0,Y 118.368,Z 878.939,A -85,B 0,C 180,E1 -27207.038,E2 -27207.038} C_VEL
LIN {X 0,Y 119.054,Z 878.719,A -85,B 0,C 180,E1 -27207.678,E2 -27207.678} C_VEL
LIN {X 0,Y 119.338,Z 879.918,A -85,B 0,C 180,E1 -27208.981,E2 -27208.981} C_VEL
LIN {X 0,Y 119.483,Z 882.873,A -85,B 0,C 180,E1 -27211.451,E2 -27211.451} C_VEL
LIN {X 0,Y 118.811,Z 886.511,A -85,B 0,C 180,E1 -27213.723,E2 -27213.723} C_VEL
LIN {X 0,Y 116.627,Z 894.032,A -85,B 0,C 180,E1 -27218.207,E2 -27218.207} C_VEL
LIN {X 0,Y 115.829,Z 898.328,A -85,B 0,C 180,E1 -27221.505,E2 -27221.505} C_VEL
LIN {X 0,Y 115.415,Z 902.83,A -85,B 0,C 180,E1 -27225.543,E2 -27225.543} C_VEL
LIN {X 0,Y 109.426,Z 910.644,A -85,B 0,C 180,E1 -27230.031,E2 -27230.031} C_VEL
LIN {X 0,Y 104.042,Z 916.903,A -85,B 0,C 180,E1 -27234.95,E2 -27234.95} C_VEL
LIN {X 0,Y 99.122,Z 921.895,A -85,B 0,C 180,E1 -27240.236,E2 -27240.236} C_VEL
LIN {X 0,Y 94.845,Z 925.785,A -85,B 0,C 180,E1 -27245.941,E2 -27245.941} C_VEL
LIN {X 0,Y 91.797,Z 928.605,A -85,B 0,C 180,E1 -27252.159,E2 -27252.159} C_VEL
LIN {X 0,Y 90.316,Z 929.945,A -85,B 0,C 180,E1 -27256.492,E2 -27256.492} C_VEL
LIN {X 0,Y 88.389,Z 931.517,A -85,B 0,C 180,E1 -27265.431,E2 -27265.431} C_VEL
LIN {X 0,Y 88.22,Z 931.729,A -85,B 0,C 180,E1 -27269.992,E2 -27269.992} C_VEL
LIN {X 0,Y 89.116,Z 930.966,A -85,B 0,C 180,E1 -27279.067,E2 -27279.067} C_VEL
LIN {X 0,Y 90.298,Z 930.015,A -85,B 0,C 180,E1 -27283.494,E2 -27283.494} C_VEL
LIN {X 0,Y 91.776,Z 928.704,A -85,B 0,C 180,E1 -27287.828,E2 -27287.828} C_VEL
LIN {X 0,Y 94.819,Z 925.915,A -85,B 0,C 180,E1 -27294.049,E2 -27294.049} C_VEL
LIN {X 0,Y 99.101,Z 922.062,A -85,B 0,C 180,E1 -27299.755,E2 -27299.755} C_VEL
LIN {X 0,Y 104.012,Z 917.124,A -85,B 0,C 180,E1 -27305.044,E2 -27305.044} C_VEL
LIN {X 0,Y 110.346,Z 909.738,A -85,B 0,C 180,E1 -27310.746,E2 -27310.746} C_VEL
LIN {X 0,Y 115.469,Z 903.159,A -85,B 0,C 180,E1 -27314.413,E2 -27314.413} C_VEL
LIN {X 0,Y 115.977,Z 897.669,A -85,B 0,C 180,E1 -27319.351,E2 -27319.351} C_VEL
LIN {X 0,Y 115.914,Z 892.498,A -85,B 0,C 180,E1 -27324.155,E2 -27324.155} C_VEL
LIN {X 0,Y 115.31,Z 887.271,A -85,B 0,C 180,E1 -27329.596,E2 -27329.596} C_VEL
LIN {X 0,Y 114.53,Z 883.146,A -85,B 0,C 180,E1 -27334.561,E2 -27334.561} C_VEL
LIN {X 0,Y 113.631,Z 879.434,A -85,B 0,C 180,E1 -27340.112,E2 -27340.112} C_VEL
LIN {X 0,Y 112.981,Z 876.622,A -85,B 0,C 180,E1 -27345.592,E2 -27345.592} C_VEL
LIN {X 0,Y 112.734,Z 875.276,A -85,B 0,C 180,E1 -27349.221,E2 -27349.221} C_VEL
LIN {X 0,Y 112.641,Z 874.055,A -85,B 0,C 180,E1 -27356.522,E2 -27356.522} C_VEL
LIN {X 0,Y 113.001,Z 873.911,A -85,B 0,C 180,E1 -27360,E2 -27360} C_VEL
LIN {X 0,Y 113.201,Z 877.324,A -85,B 0,C 180,E1 -27367.133,E2 -27367.133} C_VEL
LIN {X 0,Y 113.702,Z 879.546,A -85,B 0,C 180,E1 -27370.686,E2 -27370.686} C_VEL
LIN {X 0,Y 114.834,Z 886.694,A -85,B 0,C 180,E1 -27378.284,E2 -27378.284} C_VEL
LIN {X 0,Y 115.489,Z 891.576,A -85,B 0,C 180,E1 -27382.355,E2 -27382.355} C_VEL
LIN {X 0,Y 116.074,Z 898.061,A -85,B 0,C 180,E1 -27387.007,E2 -27387.007} C_VEL
LIN {X 0,Y 116.299,Z 903.762,A -85,B 0,C 180,E1 -27390.701,E2 -27390.701} C_VEL
LIN {X 0,Y 115.675,Z 906.093,A -85,B 0,C 180,E1 -27391.738,E2 -27391.738} C_VEL
LIN {X 0,Y 111.329,Z 916.783,A -85,B 0,C 180,E1 -27396.413,E2 -27396.413} C_VEL
LIN {X 0,Y 106.173,Z 926.873,A -85,B 0,C 180,E1 -27401.692,E2 -27401.692} C_VEL
LIN {X 0,Y 101.841,Z 934.02,A -85,B 0,C 180,E1 -27406.373,E2 -27406.373} C_VEL
LIN {X 0,Y 97.84,Z 939.896,A -85,B 0,C 180,E1 -27411.201,E2 -27411.201} C_VEL
LIN {X 0,Y 94.065,Z 944.524,A -85,B 0,C 180,E1 -27415.929,E2 -27415.929} C_VEL
LIN {X 0,Y 90.029,Z 949.07,A -85,B 0,C 180,E1 -27422.08,E2 -27422.08} C_VEL
LIN {X 0,Y 87.358,Z 952.588,A -85,B 0,C 180,E1 -27428.784,E2 -27428.784} C_VEL
LIN {X 0,Y 85.988,Z 955.133,A -85,B 0,C 180,E1 -27435.815,E2 -27435.815} C_VEL
LIN {X 0,Y 85.804,Z 956.305,A -85,B 0,C 180,E1 -27440.58,E2 -27440.58} C_VEL
LIN {X 0,Y 86.127,Z 957.078,A -85,B 0,C 180,E1 -27445.328,E2 -27445.328} C_VEL
LIN {X 0,Y 86.764,Z 957.419,A -85,B 0,C 180,E1 -27450.008,E2 -27450.008} C_VEL
LIN {X 0,Y 86.175,Z 957.065,A -85,B 0,C 180,E1 -27454.686,E2 -27454.686} C_VEL
LIN {X 0,Y 86.2,Z 955.119,A -85,B 0,C 180,E1 -27464.166,E2 -27464.166} C_VEL
LIN {X 0,Y 87.831,Z 952.589,A -85,B 0,C 180,E1 -27471.113,E2 -27471.113} C_VEL
LIN {X 0,Y 90.83,Z 949.104,A -85,B 0,C 180,E1 -27477.67,E2 -27477.67} C_VEL
LIN {X 0,Y 95.318,Z 944.619,A -85,B 0,C 180,E1 -27483.581,E2 -27483.581} C_VEL
LIN {X 0,Y 101.055,Z 939.004,A -85,B 0,C 180,E1 -27488.758,E2 -27488.758} C_VEL
LIN {X 0,Y 104.516,Z 935.766,A -85,B 0,C 180,E1 -27491.125,E2 -27491.125} C_VEL
LIN {X 0,Y 113.465,Z 936.655,A -85,B 0,C 180,E1 -27498.02,E2 -27498.02} C_VEL
LIN {X 0,Y 116.324,Z 936.766,A -85,B 0,C 180,E1 -27499.8,E2 -27499.8} C_VEL
LIN {X 0,Y 117.234,Z 936.682,A -85,B 0,C 180,E1 -27500.569,E2 -27500.569} C_VEL
LIN {X 0,Y 107.603,Z 930.608,A -85,B 0,C 180,E1 -27506.278,E2 -27506.278} C_VEL
LIN {X 0,Y 101.62,Z 925.483,A -85,B 0,C 180,E1 -27511.045,E2 -27511.045} C_VEL
LIN {X 0,Y 95.257,Z 917.377,A -85,B 0,C 180,E1 -27518.353,E2 -27518.353} C_VEL
LIN {X 0,Y 92.306,Z 911.813,A -85,B 0,C 180,E1 -27523.41,E2 -27523.41} C_VEL
LIN {X 0,Y 90.756,Z 911.23,A -85,B 0,C 180,E1 -27526.567,E2 -27526.567} C_VEL
LIN {X 0,Y 90.516,Z 905.853,A -85,B 0,C 180,E1 -27540,E2 -27540} C_VEL
LIN {X 0,Y 92.136,Z 903.37,A -85,B 0,C 180,E1 -27544.375,E2 -27544.375} C_VEL
LIN {X 0,Y 93.562,Z 901.633,A -85,B 0,C 180,E1 -27548.641,E2 -27548.641} C_VEL
LIN {X 0,Y 95.131,Z 900.09,A -85,B 0,C 180,E1 -27551.337,E2 -27551.337} C_VEL
LIN {X 0,Y 97.816,Z 897.668,A -85,B 0,C 180,E1 -27554.565,E2 -27554.565} C_VEL
LIN {X 0,Y 100.576,Z 895.68,A -85,B 0,C 180,E1 -27558.328,E2 -27558.328} C_VEL
LIN {X 0,Y 106.747,Z 890.975,A -85,B 0,C 180,E1 -27563.268,E2 -27563.268} C_VEL
LIN {X 0,Y 110.71,Z 888.501,A -85,B 0,C 180,E1 -27566.383,E2 -27566.383} C_VEL
LIN {X 0,Y 113.939,Z 886.146,A -85,B 0,C 180,E1 -27568.181,E2 -27568.181} C_VEL
LIN {X 0,Y 114.93,Z 886.05,A -85,B 0,C 180,E1 -27569.289,E2 -27569.289} C_VEL
LIN {X 0,Y 115.574,Z 890.883,A -85,B 0,C 180,E1 -27574.422,E2 -27574.422} C_VEL
LIN {X 0,Y 115.837,Z 896.23,A -85,B 0,C 180,E1 -27579.57,E2 -27579.57} C_VEL
LIN {X 0,Y 115.829,Z 898.328,A -85,B 0,C 180,E1 -27581.505,E2 -27581.505} C_VEL
LIN {X 0,Y 115.173,Z 900.178,A -85,B 0,C 180,E1 -27582.755,E2 -27582.755} C_VEL
LIN {X 0,Y 112.904,Z 903.183,A -85,B 0,C 180,E1 -27584.073,E2 -27584.073} C_VEL
LIN {X 0,Y 105.61,Z 910.146,A -85,B 0,C 180,E1 -27586.633,E2 -27586.633} C_VEL
LIN {X 0,Y 104.086,Z 911.74,A -85,B 0,C 180,E1 -27587.592,E2 -27587.592} C_VEL
LIN {X 0,Y 98.375,Z 917.936,A -85,B 0,C 180,E1 -27592.601,E2 -27592.601} C_VEL
LIN {X 0,Y 93.089,Z 922.928,A -85,B 0,C 180,E1 -27598.089,E2 -27598.089} C_VEL
LIN {X 0,Y 88.477,Z 926.817,A -85,B 0,C 180,E1 -27604.086,E2 -27604.086} C_VEL
LIN {X 0,Y 85.136,Z 929.637,A -85,B 0,C 180,E1 -27610.71,E2 -27610.71} C_VEL
LIN {X 0,Y 83.501,Z 930.977,A -85,B 0,C 180,E1 -27615.366,E2 -27615.366} C_VEL
LIN {X 0,Y 81.408,Z 932.545,A -85,B 0,C 180,E1 -27625.039,E2 -27625.039} C_VEL
LIN {X 0,Y 81.204,Z 932.759,A -85,B 0,C 180,E1 -27629.991,E2 -27629.991} C_VEL
LIN {X 0,Y 82.187,Z 931.997,A -85,B 0,C 180,E1 -27639.838,E2 -27639.838} C_VEL
LIN {X 0,Y 83.483,Z 931.046,A -85,B 0,C 180,E1 -27644.62,E2 -27644.62} C_VEL
LIN {X 0,Y 85.116,Z 929.735,A -85,B 0,C 180,E1 -27649.277,E2 -27649.277} C_VEL
LIN {X 0,Y 88.45,Z 926.945,A -85,B 0,C 180,E1 -27655.904,E2 -27655.904} C_VEL
LIN {X 0,Y 93.068,Z 923.092,A -85,B 0,C 180,E1 -27661.901,E2 -27661.901} C_VEL
LIN {X 0,Y 98.344,Z 918.154,A -85,B 0,C 180,E1 -27667.394,E2 -27667.394} C_VEL
LIN {X 0,Y 105.122,Z 910.768,A -85,B 0,C 180,E1 -27673.247,E2 -27673.247} C_VEL
LIN {X 0,Y 109.387,Z 905.658,A -85,B 0,C 180,E1 -27676.264,E2 -27676.264} C_VEL
LIN {X 0,Y 110.076,Z 902.899,A -85,B 0,C 180,E1 -27678.821,E2 -27678.821} C_VEL
LIN {X 0,Y 110.484,Z 898.376,A -85,B 0,C 180,E1 -27683.395,E2 -27683.395} C_VEL
LIN {X 0,Y 110.48,Z 893.887,A -85,B 0,C 180,E1 -27688.309,E2 -27688.309} C_VEL
LIN {X 0,Y 110.176,Z 889.741,A -85,B 0,C 180,E1 -27693.479,E2 -27693.479} C_VEL
LIN {X 0,Y 109.631,Z 885.915,A -85,B 0,C 180,E1 -27699.354,E2 -27699.354} C_VEL
LIN {X 0,Y 109.262,Z 883.032,A -85,B 0,C 180,E1 -27705.09,E2 -27705.09} C_VEL
LIN {X 0,Y 109.149,Z 881.614,A -85,B 0,C 180,E1 -27708.862,E2 -27708.862} C_VEL
LIN {X 0,Y 109.289,Z 880.357,A -85,B 0,C 180,E1 -27716.313,E2 -27716.313} C_VEL
LIN {X 0,Y 109.647,Z 880.332,A -85,B 0,C 180,E1 -27720,E2 -27720} C_VEL
LIN {X 0,Y 109.738,Z 883.85,A -85,B 0,C 180,E1 -27727.359,E2 -27727.359} C_VEL
LIN {X 0,Y 109.92,Z 884.947,A -85,B 0,C 180,E1 -27729.198,E2 -27729.198} C_VEL
LIN {X 0,Y 110.515,Z 891.266,A -85,B 0,C 180,E1 -27736.63,E2 -27736.63} C_VEL
LIN {X 0,Y 110.788,Z 896.646,A -85,B 0,C 180,E1 -27741.393,E2 -27741.393} C_VEL
LIN {X 0,Y 110.91,Z 902.093,A -85,B 0,C 180,E1 -27745.628,E2 -27745.628} C_VEL
LIN {X 0,Y 110.791,Z 906.986,A -85,B 0,C 180,E1 -27749.1,E2 -27749.1} C_VEL
LIN {X 0,Y 106.892,Z 915.643,A -85,B 0,C 180,E1 -27753.053,E2 -27753.053} C_VEL
LIN {X 0,Y 102.241,Z 924.096,A -85,B 0,C 180,E1 -27757.498,E2 -27757.498} C_VEL
LIN {X 0,Y 97.517,Z 931.621,A -85,B 0,C 180,E1 -27762.39,E2 -27762.39} C_VEL
LIN {X 0,Y 92.324,Z 938.714,A -85,B 0,C 180,E1 -27768.246,E2 -27768.246} C_VEL
LIN {X 0,Y 88.031,Z 943.663,A -85,B 0,C 180,E1 -27773.549,E2 -27773.549} C_VEL
LIN {X 0,Y 83.766,Z 948.019,A -85,B 0,C 180,E1 -27779.785,E2 -27779.785} C_VEL
LIN {X 0,Y 80.707,Z 951.535,A -85,B 0,C 180,E1 -27786.94,E2 -27786.94} C_VEL
LIN {X 0,Y 79.045,Z 954.08,A -85,B 0,C 180,E1 -27794.54,E2 -27794.54} C_VEL
LIN {X 0,Y 78.767,Z 955.256,A -85,B 0,C 180,E1 -27799.73,E2 -27799.73} C_VEL
LIN {X 0,Y 79.018,Z 956.03,A -85,B 0,C 180,E1 -27804.906,E2 -27804.906} C_VEL
LIN {X 0,Y 79.675,Z 956.378,A -85,B 0,C 180,E1 -27810.009,E2 -27810.009} C_VEL
LIN {X 0,Y 79.068,Z 956.018,A -85,B 0,C 180,E1 -27815.109,E2 -27815.109} C_VEL
LIN {X 0,Y 79.303,Z 954.071,A -85,B 0,C 180,E1 -27825.428,E2 -27825.428} C_VEL
LIN {X 0,Y 81.209,Z 951.54,A -85,B 0,C 180,E1 -27832.929,E2 -27832.929} C_VEL
LIN {X 0,Y 84.605,Z 948.061,A -85,B 0,C 180,E1 -27839.904,E2 -27839.904} C_VEL
LIN {X 0,Y 89.502,Z 943.577,A -85,B 0,C 180,E1 -27846.09,E2 -27846.09} C_VEL
LIN {X 0,Y 95.667,Z 937.969,A -85,B 0,C 180,E1 -27851.398,E2 -27851.398} C_VEL
LIN {X 0,Y 101.07,Z 933.087,A -85,B 0,C 180,E1 -27854.806,E2 -27854.806} C_VEL
LIN {X 0,Y 106.837,Z 933.892,A -85,B 0,C 180,E1 -27859.163,E2 -27859.163} C_VEL
LIN {X 0,Y 108.005,Z 933.879,A -85,B 0,C 180,E1 -27860.241,E2 -27860.241} C_VEL
LIN {X 0,Y 97.543,Z 925.918,A -85,B 0,C 180,E1 -27867.291,E2 -27867.291} C_VEL
LIN {X 0,Y 92.394,Z 920.509,A -85,B 0,C 180,E1 -27872.232,E2 -27872.232} C_VEL
LIN {X 0,Y 88.93,Z 919.397,A -85,B 0,C 180,E1 -27876.725,E2 -27876.725} C_VEL
LIN {X 0,Y 87.276,Z 917.575,A -85,B 0,C 180,E1 -27881.21,E2 -27881.21} C_VEL
LIN {X 0,Y 84.966,Z 914.446,A -85,B 0,C 180,E1 -27890.478,E2 -27890.478} C_VEL
LIN {X 0,Y 85.317,Z 910.969,A -85,B 0,C 180,E1 -27900,E2 -27900} C_VEL
LIN {X 0,Y 86.888,Z 908.743,A -85,B 0,C 180,E1 -27904.64,E2 -27904.64} C_VEL
LIN {X 0,Y 90.987,Z 904.782,A -85,B 0,C 180,E1 -27913.399,E2 -27913.399} C_VEL
LIN {X 0,Y 94.377,Z 902.143,A -85,B 0,C 180,E1 -27917.33,E2 -27917.33} C_VEL
LIN {X 0,Y 98.345,Z 899.597,A -85,B 0,C 180,E1 -27921.701,E2 -27921.701} C_VEL
LIN {X 0,Y 103.83,Z 895.845,A -85,B 0,C 180,E1 -27925.616,E2 -27925.616} C_VEL
LIN {X 0,Y 106.387,Z 894.429,A -85,B 0,C 180,E1 -27927.544,E2 -27927.544} C_VEL
LIN {X 0,Y 110.265,Z 892.802,A -85,B 0,C 180,E1 -27930.657,E2 -27930.657} C_VEL
LIN {X 0,Y 110.338,Z 896.651,A -85,B 0,C 180,E1 -27934.978,E2 -27934.978} C_VEL
LIN {X 0,Y 110.075,Z 901.832,A -85,B 0,C 180,E1 -27940.388,E2 -27940.388} C_VEL
LIN {X 0,Y 109.482,Z 905.334,A -85,B 0,C 180,E1 -27943.799,E2 -27943.799} C_VEL
LIN {X 0,Y 104.086,Z 911.74,A -85,B 0,C 180,E1 -27947.592,E2 -27947.592} C_VEL
LIN {X 0,Y 100.808,Z 914.955,A -85,B 0,C 180,E1 -27949.689,E2 -27949.689} C_VEL
LIN {X 0,Y 94.023,Z 919.919,A -85,B 0,C 180,E1 -27952.799,E2 -27952.799} C_VEL
LIN {X 0,Y 87.175,Z 924.294,A -85,B 0,C 180,E1 -27956.466,E2 -27956.466} C_VEL
LIN {X 0,Y 83.951,Z 926.477,A -85,B 0,C 180,E1 -27959.455,E2 -27959.455} C_VEL
LIN {X 0,Y 80.823,Z 928.883,A -85,B 0,C 180,E1 -27964.219,E2 -27964.219} C_VEL
LIN {X 0,Y 78.539,Z 930.669,A -85,B 0,C 180,E1 -27969.017,E2 -27969.017} C_VEL
LIN {X 0,Y 76.723,Z 932.009,A -85,B 0,C 180,E1 -27974.04,E2 -27974.04} C_VEL
LIN {X 0,Y 74.429,Z 933.574,A -85,B 0,C 180,E1 -27984.572,E2 -27984.572} C_VEL
LIN {X 0,Y 74.188,Z 933.789,A -85,B 0,C 180,E1 -27989.99,E2 -27989.99} C_VEL
LIN {X 0,Y 75.276,Z 933.028,A -85,B 0,C 180,E1 -28000.752,E2 -28000.752} C_VEL
LIN {X 0,Y 76.706,Z 932.077,A -85,B 0,C 180,E1 -28005.944,E2 -28005.944} C_VEL
LIN {X 0,Y 78.518,Z 930.766,A -85,B 0,C 180,E1 -28010.969,E2 -28010.969} C_VEL
LIN {X 0,Y 82.188,Z 927.976,A -85,B 0,C 180,E1 -28018.044,E2 -28018.044} C_VEL
LIN {X 0,Y 87.183,Z 924.122,A -85,B 0,C 180,E1 -28024.342,E2 -28024.342} C_VEL
LIN {X 0,Y 92.862,Z 919.184,A -85,B 0,C 180,E1 -28030.027,E2 -28030.027} C_VEL
LIN {X 0,Y 100.12,Z 911.797,A -85,B 0,C 180,E1 -28036.003,E2 -28036.003} C_VEL
LIN {X 0,Y 103.476,Z 908.013,A -85,B 0,C 180,E1 -28038.329,E2 -28038.329} C_VEL
LIN {X 0,Y 104.264,Z 906.081,A -85,B 0,C 180,E1 -28040.172,E2 -28040.172} C_VEL
LIN {X 0,Y 105.018,Z 901.416,A -85,B 0,C 180,E1 -28045.492,E2 -28045.492} C_VEL
LIN {X 0,Y 105.313,Z 897.649,A -85,B 0,C 180,E1 -28050.16,E2 -28050.16} C_VEL
LIN {X 0,Y 105.325,Z 894.339,A -85,B 0,C 180,E1 -28054.84,E2 -28054.84} C_VEL
LIN {X 0,Y 105.198,Z 891.063,A -85,B 0,C 180,E1 -28060.486,E2 -28060.486} C_VEL
LIN {X 0,Y 105.139,Z 889.213,A -85,B 0,C 180,E1 -28064.491,E2 -28064.491} C_VEL
LIN {X 0,Y 105.194,Z 887.795,A -85,B 0,C 180,E1 -28068.438,E2 -28068.438} C_VEL
LIN {X 0,Y 105.286,Z 886.935,A -85,B 0,C 180,E1 -28072.328,E2 -28072.328} C_VEL
LIN {X 0,Y 105.615,Z 886.449,A -85,B 0,C 180,E1 -28076.395,E2 -28076.395} C_VEL
LIN {X 0,Y 105.947,Z 886.555,A -85,B 0,C 180,E1 -28080,E2 -28080} C_VEL
LIN {X 0,Y 105.867,Z 890.184,A -85,B 0,C 180,E1 -28087.63,E2 -28087.63} C_VEL
LIN {X 0,Y 105.816,Z 894.683,A -85,B 0,C 180,E1 -28093.442,E2 -28093.442} C_VEL
LIN {X 0,Y 105.993,Z 896.242,A -85,B 0,C 180,E1 -28095.38,E2 -28095.38} C_VEL
LIN {X 0,Y 105.86,Z 901.627,A -85,B 0,C 180,E1 -28100.502,E2 -28100.502} C_VEL
LIN {X 0,Y 105.489,Z 907.865,A -85,B 0,C 180,E1 -28105.661,E2 -28105.661} C_VEL
LIN {X 0,Y 105.35,Z 909.26,A -85,B 0,C 180,E1 -28106.763,E2 -28106.763} C_VEL
LIN {X 0,Y 102.811,Z 914.491,A -85,B 0,C 180,E1 -28109.375,E2 -28109.375} C_VEL
LIN {X 0,Y 98.681,Z 921.671,A -85,B 0,C 180,E1 -28113.208,E2 -28113.208} C_VEL
LIN {X 0,Y 92.662,Z 930.53,A -85,B 0,C 180,E1 -28118.989,E2 -28118.989} C_VEL
LIN {X 0,Y 86.992,Z 937.64,A -85,B 0,C 180,E1 -28125.029,E2 -28125.029} C_VEL
LIN {X 0,Y 82.758,Z 942.248,A -85,B 0,C 180,E1 -28130.128,E2 -28130.128} C_VEL
LIN {X 0,Y 77.665,Z 946.969,A -85,B 0,C 180,E1 -28137.127,E2 -28137.127} C_VEL
LIN {X 0,Y 74.149,Z 950.481,A -85,B 0,C 180,E1 -28144.764,E2 -28144.764} C_VEL
LIN {X 0,Y 72.162,Z 953.028,A -85,B 0,C 180,E1 -28153.022,E2 -28153.022} C_VEL
LIN {X 0,Y 71.756,Z 954.209,A -85,B 0,C 180,E1 -28158.714,E2 -28158.714} C_VEL
LIN {X 0,Y 71.918,Z 954.984,A -85,B 0,C 180,E1 -28164.402,E2 -28164.402} C_VEL
LIN {X 0,Y 72.579,Z 955.336,A -85,B 0,C 180,E1 -28170.01,E2 -28170.01} C_VEL
LIN {X 0,Y 71.972,Z 954.971,A -85,B 0,C 180,E1 -28175.614,E2 -28175.614} C_VEL
LIN {X 0,Y 72.444,Z 953.022,A -85,B 0,C 180,E1 -28186.93,E2 -28186.93} C_VEL
LIN {X 0,Y 74.687,Z 950.492,A -85,B 0,C 180,E1 -28195.062,E2 -28195.062} C_VEL
LIN {X 0,Y 78.533,Z 947.018,A -85,B 0,C 180,E1 -28202.486,E2 -28202.486} C_VEL
LIN {X 0,Y 83.887,Z 942.537,A -85,B 0,C 180,E1 -28208.938,E2 -28208.938} C_VEL
LIN {X 0,Y 90.506,Z 936.934,A -85,B 0,C 180,E1 -28214.347,E2 -28214.347} C_VEL
LIN {X 0,Y 97.996,Z 930.34,A -85,B 0,C 180,E1 -28218.646,E2 -28218.646} C_VEL
LIN {X 0,Y 98.296,Z 930.395,A -85,B 0,C 180,E1 -28218.861,E2 -28218.861} C_VEL
LIN {X 0,Y 98.555,Z 930.014,A -85,B 0,C 180,E1 -28220.075,E2 -28220.075} C_VEL
LIN {X 0,Y 95.908,Z 928.049,A -85,B 0,C 180,E1 -28221.809,E2 -28221.809} C_VEL
LIN {X 0,Y 93.837,Z 927.789,A -85,B 0,C 180,E1 -28223.19,E2 -28223.19} C_VEL
LIN {X 0,Y 89.927,Z 926.641,A -85,B 0,C 180,E1 -28226.834,E2 -28226.834} C_VEL
LIN {X 0,Y 87.015,Z 924.962,A -85,B 0,C 180,E1 -28231.013,E2 -28231.013} C_VEL
LIN {X 0,Y 83.882,Z 923.887,A -85,B 0,C 180,E1 -28235.234,E2 -28235.234} C_VEL
LIN {X 0,Y 79.837,Z 915.795,A -85,B 0,C 180,E1 -28260,E2 -28260} C_VEL
LIN {X 0,Y 85.704,Z 909.942,A -85,B 0,C 180,E1 -28274.242,E2 -28274.242} C_VEL
LIN {X 0,Y 90.952,Z 906.351,A -85,B 0,C 180,E1 -28280.348,E2 -28280.348} C_VEL
LIN {X 0,Y 94.618,Z 904.263,A -85,B 0,C 180,E1 -28283.993,E2 -28283.993} C_VEL
LIN {X 0,Y 101.873,Z 899.938,A -85,B 0,C 180,E1 -28288.876,E2 -28288.876} C_VEL
LIN {X 0,Y 104.017,Z 898.947,A -85,B 0,C 180,E1 -28290.447,E2 -28290.447} C_VEL
LIN {X 0,Y 104.98,Z 899.462,A -85,B 0,C 180,E1 -28292.383,E2 -28292.383} C_VEL
LIN {X 0,Y 104.439,Z 904.431,A -85,B 0,C 180,E1 -28298.242,E2 -28298.242} C_VEL
LIN {X 0,Y 103.622,Z 907.681,A -85,B 0,C 180,E1 -28301.74,E2 -28301.74} C_VEL
LIN {X 0,Y 97.168,Z 914.729,A -85,B 0,C 180,E1 -28306.327,E2 -28306.327} C_VEL
LIN {X 0,Y 90.974,Z 920.731,A -85,B 0,C 180,E1 -28311.819,E2 -28311.819} C_VEL
LIN {X 0,Y 85.406,Z 925.362,A -85,B 0,C 180,E1 -28317.655,E2 -28317.655} C_VEL
LIN {X 0,Y 83.951,Z 926.477,A -85,B 0,C 180,E1 -28319.455,E2 -28319.455} C_VEL
LIN {X 0,Y 80.959,Z 928.463,A -85,B 0,C 180,E1 -28322.728,E2 -28322.728} C_VEL
LIN {X 0,Y 75.094,Z 931.333,A -85,B 0,C 180,E1 -28328.222,E2 -28328.222} C_VEL
LIN {X 0,Y 70.782,Z 933.066,A -85,B 0,C 180,E1 -28333.286,E2 -28333.286} C_VEL
LIN {X 0,Y 68.567,Z 933.946,A -85,B 0,C 180,E1 -28337.743,E2 -28337.743} C_VEL
LIN {X 0,Y 68.146,Z 934.135,A -85,B 0,C 180,E1 -28339.351,E2 -28339.351} C_VEL
LIN {X 0,Y 67.171,Z 934.819,A -85,B 0,C 180,E1 -28349.989,E2 -28349.989} C_VEL
LIN {X 0,Y 68.387,Z 934.059,A -85,B 0,C 180,E1 -28361.85,E2 -28361.85} C_VEL
LIN {X 0,Y 69.977,Z 933.108,A -85,B 0,C 180,E1 -28367.525,E2 -28367.525} C_VEL
LIN {X 0,Y 72.002,Z 931.796,A -85,B 0,C 180,E1 -28372.97,E2 -28372.97} C_VEL
LIN {X 0,Y 76.059,Z 929.006,A -85,B 0,C 180,E1 -28380.533,E2 -28380.533} C_VEL
LIN {X 0,Y 81.479,Z 925.152,A -85,B 0,C 180,E1 -28387.13,E2 -28387.13} C_VEL
LIN {X 0,Y 87.599,Z 920.214,A -85,B 0,C 180,E1 -28392.984,E2 -28392.984} C_VEL
LIN {X 0,Y 95.372,Z 912.827,A -85,B 0,C 180,E1 -28399.041,E2 -28399.041} C_VEL
LIN {X 0,Y 97.734,Z 910.36,A -85,B 0,C 180,E1 -28400.614,E2 -28400.614} C_VEL
LIN {X 0,Y 98.464,Z 909.155,A -85,B 0,C 180,E1 -28401.721,E2 -28401.721} C_VEL
LIN {X 0,Y 99.596,Z 904.42,A -85,B 0,C 180,E1 -28407.849,E2 -28407.849} C_VEL
LIN {X 0,Y 100.149,Z 900.897,A -85,B 0,C 180,E1 -28412.861,E2 -28412.861} C_VEL
LIN {X 0,Y 100.418,Z 898.208,A -85,B 0,C 180,E1 -28417.338,E2 -28417.338} C_VEL
LIN {X 0,Y 100.625,Z 895.218,A -85,B 0,C 180,E1 -28423.777,E2 -28423.777} C_VEL
LIN {X 0,Y 100.89,Z 893.755,A -85,B 0,C 180,E1 -28427.937,E2 -28427.937} C_VEL
LIN {X 0,Y 101.119,Z 892.836,A -85,B 0,C 180,E1 -28432.01,E2 -28432.01} C_VEL
LIN {X 0,Y 101.536,Z 892.321,A -85,B 0,C 180,E1 -28436.031,E2 -28436.031} C_VEL
LIN {X 0,Y 101.881,Z 892.563,A -85,B 0,C 180,E1 -28440,E2 -28440} C_VEL
LIN {X 0,Y 101.592,Z 894.749,A -85,B 0,C 180,E1 -28444.977,E2 -28444.977} C_VEL
LIN {X 0,Y 101.507,Z 896.424,A -85,B 0,C 180,E1 -28447.959,E2 -28447.959} C_VEL
LIN {X 0,Y 101.15,Z 901.758,A -85,B 0,C 180,E1 -28454.896,E2 -28454.896} C_VEL
LIN {X 0,Y 100.602,Z 907.237,A -85,B 0,C 180,E1 -28460.444,E2 -28460.444} C_VEL
LIN {X 0,Y 100.015,Z 911.28,A -85,B 0,C 180,E1 -28464.025,E2 -28464.025} C_VEL
LIN {X 0,Y 99.56,Z 912.677,A -85,B 0,C 180,E1 -28465.058,E2 -28465.058} C_VEL
LIN {X 0,Y 94.686,Z 920.544,A -85,B 0,C 180,E1 -28469.309,E2 -28469.309} C_VEL
LIN {X 0,Y 88.015,Z 929.574,A -85,B 0,C 180,E1 -28475.3,E2 -28475.3} C_VEL
LIN {X 0,Y 81.935,Z 936.557,A -85,B 0,C 180,E1 -28481.378,E2 -28481.378} C_VEL
LIN {X 0,Y 76.894,Z 941.608,A -85,B 0,C 180,E1 -28487.249,E2 -28487.249} C_VEL
LIN {X 0,Y 71.767,Z 945.921,A -85,B 0,C 180,E1 -28494.029,E2 -28494.029} C_VEL
LIN {X 0,Y 67.73,Z 949.429,A -85,B 0,C 180,E1 -28502.177,E2 -28502.177} C_VEL
LIN {X 0,Y 65.339,Z 951.976,A -85,B 0,C 180,E1 -28511.186,E2 -28511.186} C_VEL
LIN {X 0,Y 64.743,Z 953.19,A -85,B 0,C 180,E1 -28517.679,E2 -28517.679} C_VEL
LIN {X 0,Y 64.829,Z 953.937,A -85,B 0,C 180,E1 -28523.788,E2 -28523.788} C_VEL
LIN {X 0,Y 65.478,Z 954.294,A -85,B 0,C 180,E1 -28530.011,E2 -28530.011} C_VEL
LIN {X 0,Y 64.887,Z 953.925,A -85,B 0,C 180,E1 -28536.229,E2 -28536.229} C_VEL
LIN {X 0,Y 65.673,Z 951.978,A -85,B 0,C 180,E1 -28548.737,E2 -28548.737} C_VEL
LIN {X 0,Y 68.298,Z 949.445,A -85,B 0,C 180,E1 -28557.596,E2 -28557.596} C_VEL
LIN {X 0,Y 72.646,Z 945.975,A -85,B 0,C 180,E1 -28565.494,E2 -28565.494} C_VEL
LIN {X 0,Y 78.513,Z 941.498,A -85,B 0,C 180,E1 -28572.183,E2 -28572.183} C_VEL
LIN {X 0,Y 85.613,Z 935.899,A -85,B 0,C 180,E1 -28577.642,E2 -28577.642} C_VEL
LIN {X 0,Y 88.179,Z 933.738,A -85,B 0,C 180,E1 -28579.227,E2 -28579.227} C_VEL
LIN {X 0,Y 89.285,Z 931.893,A -85,B 0,C 180,E1 -28580.971,E2 -28580.971} C_VEL
LIN {X 0,Y 85.134,Z 930.779,A -85,B 0,C 180,E1 -28584.699,E2 -28584.699} C_VEL
LIN {X 0,Y 81.657,Z 929.093,A -85,B 0,C 180,E1 -28589.409,E2 -28589.409} C_VEL
LIN {X 0,Y 78.681,Z 928.074,A -85,B 0,C 180,E1 -28593.474,E2 -28593.474} C_VEL
LIN {X 0,Y 74.119,Z 920.289,A -85,B 0,C 180,E1 -28620,E2 -28620} C_VEL
LIN {X 0,Y 81.827,Z 913.654,A -85,B 0,C 180,E1 -28637.494,E2 -28637.494} C_VEL
LIN {X 0,Y 87.628,Z 910.255,A -85,B 0,C 180,E1 -28643.642,E2 -28643.642} C_VEL
LIN {X 0,Y 91.897,Z 908.057,A -85,B 0,C 180,E1 -28647.314,E2 -28647.314} C_VEL
LIN {X 0,Y 97.039,Z 905.277,A -85,B 0,C 180,E1 -28650.463,E2 -28650.463} C_VEL
LIN {X 0,Y 99.445,Z 904.125,A -85,B 0,C 180,E1 -28652.005,E2 -28652.005} C_VEL
LIN {X 0,Y 98.403,Z 908.875,A -85,B 0,C 180,E1 -28658.211,E2 -28658.211} C_VEL
LIN {X 0,Y 97.852,Z 910.037,A -85,B 0,C 180,E1 -28659.447,E2 -28659.447} C_VEL
LIN {X 0,Y 90.978,Z 916.944,A -85,B 0,C 180,E1 -28664.23,E2 -28664.23} C_VEL
LIN {X 0,Y 85.563,Z 921.764,A -85,B 0,C 180,E1 -28668.91,E2 -28668.91} C_VEL
LIN {X 0,Y 79.573,Z 926.392,A -85,B 0,C 180,E1 -28674.953,E2 -28674.953} C_VEL
LIN {X 0,Y 74.56,Z 929.915,A -85,B 0,C 180,E1 -28681.871,E2 -28681.871} C_VEL
LIN {X 0,Y 72.023,Z 931.701,A -85,B 0,C 180,E1 -28687.015,E2 -28687.015} C_VEL
LIN {X 0,Y 69.994,Z 933.041,A -85,B 0,C 180,E1 -28692.458,E2 -28692.458} C_VEL
LIN {X 0,Y 68.146,Z 934.135,A -85,B 0,C 180,E1 -28699.351,E2 -28699.351} C_VEL
LIN {X 0,Y 66.743,Z 934.727,A -85,B 0,C 180,E1 -28704.213,E2 -28704.213} C_VEL
LIN {X 0,Y 63.634,Z 935.296,A -85,B 0,C 180,E1 -28712.491,E2 -28712.491} C_VEL
LIN {X 0,Y 61.949,Z 935.286,A -85,B 0,C 180,E1 -28719.598,E2 -28719.598} C_VEL
LIN {X 0,Y 62.056,Z 934.85,A -85,B 0,C 180,E1 -28725.06,E2 -28725.06} C_VEL
LIN {X 0,Y 62.464,Z 934.543,A -85,B 0,C 180,E1 -28726.826,E2 -28726.826} C_VEL
LIN {X 0,Y 65.591,Z 932.827,A -85,B 0,C 180,E1 -28735.366,E2 -28735.366} C_VEL
LIN {X 0,Y 70.099,Z 930.037,A -85,B 0,C 180,E1 -28743.451,E2 -28743.451} C_VEL
LIN {X 0,Y 75.997,Z 926.182,A -85,B 0,C 180,E1 -28750.328,E2 -28750.328} C_VEL
LIN {X 0,Y 82.599,Z 921.243,A -85,B 0,C 180,E1 -28756.308,E2 -28756.308} C_VEL
LIN {X 0,Y 89.688,Z 915.052,A -85,B 0,C 180,E1 -28761.578,E2 -28761.578} C_VEL
LIN {X 0,Y 92.175,Z 912.661,A -85,B 0,C 180,E1 -28763.172,E2 -28763.172} C_VEL
LIN {X 0,Y 92.939,Z 911.513,A -85,B 0,C 180,E1 -28764.366,E2 -28764.366} C_VEL
LIN {X 0,Y 93.857,Z 908.776,A -85,B 0,C 180,E1 -28768.388,E2 -28768.388} C_VEL
LIN {X 0,Y 94.808,Z 905.459,A -85,B 0,C 180,E1 -28773.591,E2 -28773.591} C_VEL
LIN {X 0,Y 95.39,Z 902.888,A -85,B 0,C 180,E1 -28778.384,E2 -28778.384} C_VEL
LIN {X 0,Y 95.757,Z 901.005,A -85,B 0,C 180,E1 -28782.927,E2 -28782.927} C_VEL
LIN {X 0,Y 96.181,Z 899.479,A -85,B 0,C 180,E1 -28787.337,E2 -28787.337} C_VEL
LIN {X 0,Y 96.626,Z 898.516,A -85,B 0,C 180,E1 -28791.635,E2 -28791.635} C_VEL
LIN {X 0,Y 97.142,Z 897.974,A -85,B 0,C 180,E1 -28795.851,E2 -28795.851} C_VEL
LIN {X 0,Y 97.44,Z 898.331,A -85,B 0,C 180,E1 -28800,E2 -28800} C_VEL
LIN {X 0,Y 96.946,Z 901.174,A -85,B 0,C 180,E1 -28806.243,E2 -28806.243} C_VEL
LIN {X 0,Y 96.289,Z 905.528,A -85,B 0,C 180,E1 -28812.648,E2 -28812.648} C_VEL
LIN {X 0,Y 95.391,Z 910.465,A -85,B 0,C 180,E1 -28818.245,E2 -28818.245} C_VEL
LIN {X 0,Y 94.584,Z 914.056,A -85,B 0,C 180,E1 -28821.809,E2 -28821.809} C_VEL
LIN {X 0,Y 93.548,Z 915.937,A -85,B 0,C 180,E1 -28823.074,E2 -28823.074} C_VEL
LIN {X 0,Y 87.506,Z 924.101,A -85,B 0,C 180,E1 -28827.957,E2 -28827.957} C_VEL
LIN {X 0,Y 80.577,Z 932.099,A -85,B 0,C 180,E1 -28834.062,E2 -28834.062} C_VEL
LIN {X 0,Y 74.093,Z 938.494,A -85,B 0,C 180,E1 -28840.655,E2 -28840.655} C_VEL
LIN {X 0,Y 70.005,Z 941.984,A -85,B 0,C 180,E1 -28845.368,E2 -28845.368} C_VEL
LIN {X 0,Y 64.388,Z 946.171,A -85,B 0,C 180,E1 -28853.121,E2 -28853.121} C_VEL
LIN {X 0,Y 60.315,Z 949.353,A -85,B 0,C 180,E1 -28862.233,E2 -28862.233} C_VEL
LIN {X 0,Y 57.777,Z 952.107,A -85,B 0,C 180,E1 -28875.933,E2 -28875.933} C_VEL
LIN {X 0,Y 57.749,Z 952.891,A -85,B 0,C 180,E1 -28883.022,E2 -28883.022} C_VEL
LIN {X 0,Y 58.373,Z 953.25,A -85,B 0,C 180,E1 -28890.012,E2 -28890.012} C_VEL
LIN {X 0,Y 57.813,Z 952.88,A -85,B 0,C 180,E1 -28896.995,E2 -28896.995} C_VEL
LIN {X 0,Y 58.95,Z 950.928,A -85,B 0,C 180,E1 -28910.969,E2 -28910.969} C_VEL
LIN {X 0,Y 62.081,Z 948.399,A -85,B 0,C 180,E1 -28920.639,E2 -28920.639} C_VEL
LIN {X 0,Y 66.994,Z 944.932,A -85,B 0,C 180,E1 -28929.021,E2 -28929.021} C_VEL
LIN {X 0,Y 73.429,Z 940.459,A -85,B 0,C 180,E1 -28935.889,E2 -28935.889} C_VEL
LIN {X 0,Y 81.02,Z 934.86,A -85,B 0,C 180,E1 -28941.337,E2 -28941.337} C_VEL
LIN {X 0,Y 76.752,Z 933.121,A -85,B 0,C 180,E1 -28946.674,E2 -28946.674} C_VEL
LIN {X 0,Y 73.371,Z 931.926,A -85,B 0,C 180,E1 -28951.384,E2 -28951.384} C_VEL
LIN {X 0,Y 68.125,Z 924.414,A -85,B 0,C 180,E1 -28980,E2 -28980} C_VEL
LIN {X 0,Y 78.054,Z 917.077,A -85,B 0,C 180,E1 -29001.11,E2 -29001.11} C_VEL
LIN {X 0,Y 89.454,Z 911.534,A -85,B 0,C 180,E1 -29010.971,E2 -29010.971} C_VEL
LIN {X 0,Y 91.898,Z 910.36,A -85,B 0,C 180,E1 -29012.367,E2 -29012.367} C_VEL
LIN {X 0,Y 93.226,Z 910.167,A -85,B 0,C 180,E1 -29013.965,E2 -29013.965} C_VEL
LIN {X 0,Y 92.255,Z 912.375,A -85,B 0,C 180,E1 -29016.869,E2 -29016.869} C_VEL
LIN {X 0,Y 84.921,Z 919.088,A -85,B 0,C 180,E1 -29021.843,E2 -29021.843} C_VEL
LIN {X 0,Y 78.175,Z 924.461,A -85,B 0,C 180,E1 -29027.592,E2 -29027.592} C_VEL
LIN {X 0,Y 71.94,Z 928.719,A -85,B 0,C 180,E1 -29034.104,E2 -29034.104} C_VEL
LIN {X 0,Y 68.445,Z 930.948,A -85,B 0,C 180,E1 -29039.097,E2 -29039.097} C_VEL
LIN {X 0,Y 65.612,Z 932.733,A -85,B 0,C 180,E1 -29044.618,E2 -29044.618} C_VEL
LIN {X 0,Y 63.33,Z 934.073,A -85,B 0,C 180,E1 -29050.542,E2 -29050.542} C_VEL
LIN {X 0,Y 60.486,Z 935.633,A -85,B 0,C 180,E1 -29063.316,E2 -29063.316} C_VEL
LIN {X 0,Y 60.174,Z 935.846,A -85,B 0,C 180,E1 -29069.988,E2 -29069.988} C_VEL
LIN {X 0,Y 61.53,Z 935.09,A -85,B 0,C 180,E1 -29083.193,E2 -29083.193} C_VEL
LIN {X 0,Y 62.464,Z 934.543,A -85,B 0,C 180,E1 -29086.826,E2 -29086.826} C_VEL
LIN {X 0,Y 63.542,Z 933.76,A -85,B 0,C 180,E1 -29092.052,E2 -29092.052} C_VEL
LIN {X 0,Y 64.555,Z 932.144,A -85,B 0,C 180,E1 -29100.772,E2 -29100.772} C_VEL
LIN {X 0,Y 66.836,Z 929.845,A -85,B 0,C 180,E1 -29108.943,E2 -29108.943} C_VEL
LIN {X 0,Y 69.682,Z 927.887,A -85,B 0,C 180,E1 -29112.957,E2 -29112.957} C_VEL
LIN {X 0,Y 77.912,Z 922.273,A -85,B 0,C 180,E1 -29120.047,E2 -29120.047} C_VEL
LIN {X 0,Y 85.498,Z 916.081,A -85,B 0,C 180,E1 -29125.27,E2 -29125.27} C_VEL
LIN {X 0,Y 86.811,Z 914.886,A -85,B 0,C 180,E1 -29126.063,E2 -29126.063} C_VEL
LIN {X 0,Y 87.562,Z 913.847,A -85,B 0,C 180,E1 -29127.417,E2 -29127.417} C_VEL
LIN {X 0,Y 88.636,Z 911.399,A -85,B 0,C 180,E1 -29131.592,E2 -29131.592} C_VEL
LIN {X 0,Y 89.783,Z 908.561,A -85,B 0,C 180,E1 -29136.959,E2 -29136.959} C_VEL
LIN {X 0,Y 90.468,Z 906.522,A -85,B 0,C 180,E1 -29141.896,E2 -29141.896} C_VEL
LIN {X 0,Y 91.099,Z 905.003,A -85,B 0,C 180,E1 -29146.618,E2 -29146.618} C_VEL
LIN {X 0,Y 92.029,Z 903.686,A -85,B 0,C 180,E1 -29153.037,E2 -29153.037} C_VEL
LIN {X 0,Y 92.421,Z 903.411,A -85,B 0,C 180,E1 -29155.639,E2 -29155.639} C_VEL
LIN {X 0,Y 92.671,Z 903.864,A -85,B 0,C 180,E1 -29160,E2 -29160} C_VEL
LIN {X 0,Y 92.213,Z 905.7,A -85,B 0,C 180,E1 -29164.371,E2 -29164.371} C_VEL
LIN {X 0,Y 91.194,Z 909.79,A -85,B 0,C 180,E1 -29171.108,E2 -29171.108} C_VEL
LIN {X 0,Y 89.927,Z 914.339,A -85,B 0,C 180,E1 -29176.78,E2 -29176.78} C_VEL
LIN {X 0,Y 89.236,Z 916.458,A -85,B 0,C 180,E1 -29179.103,E2 -29179.103} C_VEL
LIN {X 0,Y 88.654,Z 917.548,A -85,B 0,C 180,E1 -29179.99,E2 -29179.99} C_VEL
LIN {X 0,Y 82.371,Z 925.033,A -85,B 0,C 180,E1 -29184.708,E2 -29184.708} C_VEL
LIN {X 0,Y 75.417,Z 932.202,A -85,B 0,C 180,E1 -29190.479,E2 -29190.479} C_VEL
LIN {X 0,Y 69.523,Z 937.415,A -85,B 0,C 180,E1 -29196.048,E2 -29196.048} C_VEL
LIN {X 0,Y 65.077,Z 940.928,A -85,B 0,C 180,E1 -29200.909,E2 -29200.909} C_VEL
LIN {X 0,Y 58.832,Z 945.124,A -85,B 0,C 180,E1 -29208.944,E2 -29208.944} C_VEL
LIN {X 0,Y 54.059,Z 948.298,A -85,B 0,C 180,E1 -29218.682,E2 -29218.682} C_VEL
LIN {X 0,Y 50.866,Z 951.057,A -85,B 0,C 180,E1 -29233.973,E2 -29233.973} C_VEL
LIN {X 0,Y 50.684,Z 951.845,A -85,B 0,C 180,E1 -29242.044,E2 -29242.044} C_VEL
LIN {X 0,Y 51.265,Z 952.207,A -85,B 0,C 180,E1 -29250.014,E2 -29250.014} C_VEL
LIN {X 0,Y 50.755,Z 951.835,A -85,B 0,C 180,E1 -29257.974,E2 -29257.974} C_VEL
LIN {X 0,Y 52.352,Z 949.88,A -85,B 0,C 180,E1 -29273.764,E2 -29273.764} C_VEL
LIN {X 0,Y 56.086,Z 947.356,A -85,B 0,C 180,E1 -29284.34,E2 -29284.34} C_VEL
LIN {X 0,Y 61.644,Z 943.889,A -85,B 0,C 180,E1 -29293.177,E2 -29293.177} C_VEL
LIN {X 0,Y 68.7,Z 939.421,A -85,B 0,C 180,E1 -29300.122,E2 -29300.122} C_VEL
LIN {X 0,Y 71.291,Z 937.686,A -85,B 0,C 180,E1 -29302.076,E2 -29302.076} C_VEL
LIN {X 0,Y 71.583,Z 936.615,A -85,B 0,C 180,E1 -29303.909,E2 -29303.909} C_VEL
LIN {X 0,Y 65.178,Z 934.055,A -85,B 0,C 180,E1 -29314.45,E2 -29314.45} C_VEL
LIN {X 0,Y 61.933,Z 928.18,A -85,B 0,C 180,E1 -29340,E2 -29340} C_VEL
LIN {X 0,Y 68.677,Z 923.068,A -85,B 0,C 180,E1 -29357.879,E2 -29357.879} C_VEL
LIN {X 0,Y 83.466,Z 916.36,A -85,B 0,C 180,E1 -29372.632,E2 -29372.632} C_VEL
LIN {X 0,Y 85.549,Z 915.808,A -85,B 0,C 180,E1 -29374.75,E2 -29374.75} C_VEL
LIN {X 0,Y 77.947,Z 922.066,A -85,B 0,C 180,E1 -29379.956,E2 -29379.956} C_VEL
LIN {X 0,Y 70.814,Z 927.057,A -85,B 0,C 180,E1 -29385.982,E2 -29385.982} C_VEL
LIN {X 0,Y 64.384,Z 930.946,A -85,B 0,C 180,E1 -29393.091,E2 -29393.091} C_VEL
LIN {X 0,Y 59.34,Z 933.765,A -85,B 0,C 180,E1 -29401.709,E2 -29401.709} C_VEL
LIN {X 0,Y 56.753,Z 935.105,A -85,B 0,C 180,E1 -29408.178,E2 -29408.178} C_VEL
LIN {X 0,Y 53.527,Z 936.663,A -85,B 0,C 180,E1 -29422.442,E2 -29422.442} C_VEL
LIN {X 0,Y 53.174,Z 936.874,A -85,B 0,C 180,E1 -29429.986,E2 -29429.986} C_VEL
LIN {X 0,Y 54.715,Z 936.121,A -85,B 0,C 180,E1 -29444.872,E2 -29444.872} C_VEL
LIN {X 0,Y 56.736,Z 935.17,A -85,B 0,C 180,E1 -29451.801,E2 -29451.801} C_VEL
LIN {X 0,Y 59.319,Z 933.858,A -85,B 0,C 180,E1 -29458.275,E2 -29458.275} C_VEL
LIN {X 0,Y 64.355,Z 931.067,A -85,B 0,C 180,E1 -29466.901,E2 -29466.901} C_VEL
LIN {X 0,Y 69.682,Z 927.887,A -85,B 0,C 180,E1 -29472.957,E2 -29472.957} C_VEL
LIN {X 0,Y 71.57,Z 926.508,A -85,B 0,C 180,E1 -29475.574,E2 -29475.574} C_VEL
LIN {X 0,Y 73.456,Z 924.439,A -85,B 0,C 180,E1 -29480.442,E2 -29480.442} C_VEL
LIN {X 0,Y 75.655,Z 922.056,A -85,B 0,C 180,E1 -29485.016,E2 -29485.016} C_VEL
LIN {X 0,Y 77.868,Z 920.168,A -85,B 0,C 180,E1 -29487.059,E2 -29487.059} C_VEL
LIN {X 0,Y 81.708,Z 917.109,A -85,B 0,C 180,E1 -29489.313,E2 -29489.313} C_VEL
LIN {X 0,Y 83.016,Z 915.083,A -85,B 0,C 180,E1 -29493.073,E2 -29493.073} C_VEL
LIN {X 0,Y 84.008,Z 913.27,A -85,B 0,C 180,E1 -29496.938,E2 -29496.938} C_VEL
LIN {X 0,Y 84.847,Z 911.76,A -85,B 0,C 180,E1 -29500.65,E2 -29500.65} C_VEL
LIN {X 0,Y 86.113,Z 909.623,A -85,B 0,C 180,E1 -29508.295,E2 -29508.295} C_VEL
LIN {X 0,Y 87.406,Z 908.558,A -85,B 0,C 180,E1 -29515.388,E2 -29515.388} C_VEL
LIN {X 0,Y 87.602,Z 909.124,A -85,B 0,C 180,E1 -29520,E2 -29520} C_VEL
LIN {X 0,Y 86.9,Z 911.087,A -85,B 0,C 180,E1 -29524.639,E2 -29524.639} C_VEL
LIN {X 0,Y 85.71,Z 914.431,A -85,B 0,C 180,E1 -29530.324,E2 -29530.324} C_VEL
LIN {X 0,Y 84.563,Z 917.411,A -85,B 0,C 180,E1 -29534.438,E2 -29534.438} C_VEL
LIN {X 0,Y 83.807,Z 919.188,A -85,B 0,C 180,E1 -29536.643,E2 -29536.643} C_VEL
LIN {X 0,Y 78.663,Z 924.736,A -85,B 0,C 180,E1 -29540.258,E2 -29540.258} C_VEL
LIN {X 0,Y 70.586,Z 932.208,A -85,B 0,C 180,E1 -29546.375,E2 -29546.375} C_VEL
LIN {X 0,Y 62.749,Z 938.331,A -85,B 0,C 180,E1 -29553.46,E2 -29553.46} C_VEL
LIN {X 0,Y 58.17,Z 941.386,A -85,B 0,C 180,E1 -29558.271,E2 -29558.271} C_VEL
LIN {X 0,Y 51.573,Z 945.22,A -85,B 0,C 180,E1 -29567.069,E2 -29567.069} C_VEL
LIN {X 0,Y 48.078,Z 947.247,A -85,B 0,C 180,E1 -29574.236,E2 -29574.236} C_VEL
LIN {X 0,Y 44.002,Z 950.002,A -85,B 0,C 180,E1 -29591.389,E2 -29591.389} C_VEL
LIN {X 0,Y 43.61,Z 950.795,A -85,B 0,C 180,E1 -29600.743,E2 -29600.743} C_VEL
LIN {X 0,Y 44.155,Z 951.163,A -85,B 0,C 180,E1 -29610.016,E2 -29610.016} C_VEL
LIN {X 0,Y 44.013,Z 950.2,A -85,B 0,C 180,E1 -29626.651,E2 -29626.651} C_VEL
LIN {X 0,Y 45.91,Z 948.832,A -85,B 0,C 180,E1 -29637.356,E2 -29637.356} C_VEL
LIN {X 0,Y 50.382,Z 946.313,A -85,B 0,C 180,E1 -29648.9,E2 -29648.9} C_VEL
LIN {X 0,Y 56.68,Z 942.847,A -85,B 0,C 180,E1 -29658.088,E2 -29658.088} C_VEL
LIN {X 0,Y 62.95,Z 939.264,A -85,B 0,C 180,E1 -29663.868,E2 -29663.868} C_VEL
LIN {X 0,Y 62.566,Z 938.55,A -85,B 0,C 180,E1 -29665.83,E2 -29665.83} C_VEL
LIN {X 0,Y 55.132,Z 933.071,A -85,B 0,C 180,E1 -29692.677,E2 -29692.677} C_VEL
LIN {X 0,Y 59.422,Z 928.406,A -85,B 0,C 180,E1 -29713.683,E2 -29713.683} C_VEL
LIN {X 0,Y 71.098,Z 923.085,A -85,B 0,C 180,E1 -29729.62,E2 -29729.62} C_VEL
LIN {X 0,Y 76.146,Z 921.137,A -85,B 0,C 180,E1 -29733.627,E2 -29733.627} C_VEL
LIN {X 0,Y 76.272,Z 921.153,A -85,B 0,C 180,E1 -29733.958,E2 -29733.958} C_VEL
LIN {X 0,Y 68.461,Z 926.526,A -85,B 0,C 180,E1 -29739.638,E2 -29739.638} C_VEL
LIN {X 0,Y 61.118,Z 930.784,A -85,B 0,C 180,E1 -29746.359,E2 -29746.359} C_VEL
LIN {X 0,Y 56.849,Z 933.012,A -85,B 0,C 180,E1 -29751.805,E2 -29751.805} C_VEL
LIN {X 0,Y 53.257,Z 934.798,A -85,B 0,C 180,E1 -29758.124,E2 -29758.124} C_VEL
LIN {X 0,Y 50.297,Z 936.137,A -85,B 0,C 180,E1 -29765.201,E2 -29765.201} C_VEL
LIN {X 0,Y 46.582,Z 937.693,A -85,B 0,C 180,E1 -29781.307,E2 -29781.307} C_VEL
LIN {X 0,Y 46.171,Z 937.902,A -85,B 0,C 180,E1 -29789.984,E2 -29789.984} C_VEL
LIN {X 0,Y 47.96,Z 937.151,A -85,B 0,C 180,E1 -29807.026,E2 -29807.026} C_VEL
LIN {X 0,Y 50.28,Z 936.201,A -85,B 0,C 180,E1 -29814.776,E2 -29814.776} C_VEL
LIN {X 0,Y 53.235,Z 934.889,A -85,B 0,C 180,E1 -29821.859,E2 -29821.859} C_VEL
LIN {X 0,Y 58.888,Z 932.098,A -85,B 0,C 180,E1 -29831.009,E2 -29831.009} C_VEL
LIN {X 0,Y 65.917,Z 928.242,A -85,B 0,C 180,E1 -29838.256,E2 -29838.256} C_VEL
LIN {X 0,Y 73.597,Z 923.303,A -85,B 0,C 180,E1 -29844.243,E2 -29844.243} C_VEL
LIN {X 0,Y 77.868,Z 920.168,A -85,B 0,C 180,E1 -29847.059,E2 -29847.059} C_VEL
LIN {X 0,Y 79.104,Z 919.034,A -85,B 0,C 180,E1 -29848.354,E2 -29848.354} C_VEL
LIN {X 0,Y 79.819,Z 917.884,A -85,B 0,C 180,E1 -29850.916,E2 -29850.916} C_VEL
LIN {X 0,Y 79.701,Z 917.222,A -85,B 0,C 180,E1 -29853.722,E2 -29853.722} C_VEL
LIN {X 0,Y 79.094,Z 916.137,A -85,B 0,C 180,E1 -29861.781,E2 -29861.781} C_VEL
LIN {X 0,Y 79.2,Z 915.952,A -85,B 0,C 180,E1 -29862.306,E2 -29862.306} C_VEL
LIN {X 0,Y 79.941,Z 915.102,A -85,B 0,C 180,E1 -29865.215,E2 -29865.215} C_VEL
LIN {X 0,Y 81.003,Z 914.055,A -85,B 0,C 180,E1 -29870.007,E2 -29870.007} C_VEL
LIN {X 0,Y 82.009,Z 913.45,A -85,B 0,C 180,E1 -29875.084,E2 -29875.084} C_VEL
LIN {X 0,Y 82.146,Z 914.109,A -85,B 0,C 180,E1 -29880,E2 -29880} C_VEL
LIN {X 0,Y 81.162,Z 916.227,A -85,B 0,C 180,E1 -29884.967,E2 -29884.967} C_VEL
LIN {X 0,Y 79.787,Z 919.19,A -85,B 0,C 180,E1 -29890.146,E2 -29890.146} C_VEL
LIN {X 0,Y 79.063,Z 920.527,A -85,B 0,C 180,E1 -29892.143,E2 -29892.143} C_VEL
LIN {X 0,Y 77.813,Z 922.181,A -85,B 0,C 180,E1 -29893.891,E2 -29893.891} C_VEL
LIN {X 0,Y 69.008,Z 929.994,A -85,B 0,C 180,E1 -29899.635,E2 -29899.635} C_VEL
LIN {X 0,Y 61.997,Z 935.252,A -85,B 0,C 180,E1 -29904.952,E2 -29904.952} C_VEL
LIN {X 0,Y 53.971,Z 940.359,A -85,B 0,C 180,E1 -29912.323,E2 -29912.323} C_VEL
LIN {X 0,Y 46.591,Z 944.171,A -85,B 0,C 180,E1 -29921.067,E2 -29921.067} C_VEL
LIN {X 0,Y 42.479,Z 946.197,A -85,B 0,C 180,E1 -29928.587,E2 -29928.587} C_VEL
LIN {X 0,Y 37.265,Z 948.948,A -85,B 0,C 180,E1 -29947.862,E2 -29947.862} C_VEL
LIN {X 0,Y 36.573,Z 949.746,A -85,B 0,C 180,E1 -29958.941,E2 -29958.941} C_VEL
LIN {X 0,Y 37.043,Z 950.119,A -85,B 0,C 180,E1 -29970.019,E2 -29970.019} C_VEL
LIN {X 0,Y 37.127,Z 949.239,A -85,B 0,C 180,E1 -29988.833,E2 -29988.833} C_VEL
LIN {X 0,Y 39.724,Z 947.787,A -85,B 0,C 180,E1 -30002.078,E2 -30002.078} C_VEL
LIN {X 0,Y 45.062,Z 945.266,A -85,B 0,C 180,E1 -30014.596,E2 -30014.596} C_VEL
LIN {X 0,Y 53.576,Z 941.147,A -85,B 0,C 180,E1 -30025.161,E2 -30025.161} C_VEL
LIN {X 0,Y 53.71,Z 940.069,A -85,B 0,C 180,E1 -30028.44,E2 -30028.44} C_VEL
LIN {X 0,Y 49.236,Z 934.295,A -85,B 0,C 180,E1 -30061.955,E2 -30061.955} C_VEL
LIN {X 0,Y 60.662,Z 928.34,A -85,B 0,C 180,E1 -30087.609,E2 -30087.609} C_VEL
LIN {X 0,Y 65.476,Z 926.587,A -85,B 0,C 180,E1 -30092.459,E2 -30092.459} C_VEL
LIN {X 0,Y 63.822,Z 927.781,A -85,B 0,C 180,E1 -30095.082,E2 -30095.082} C_VEL
LIN {X 0,Y 56.244,Z 931.816,A -85,B 0,C 180,E1 -30101.415,E2 -30101.415} C_VEL
LIN {X 0,Y 51.511,Z 934.044,A -85,B 0,C 180,E1 -30106.968,E2 -30106.968} C_VEL
LIN {X 0,Y 47.436,Z 935.83,A -85,B 0,C 180,E1 -30113.638,E2 -30113.638} C_VEL
LIN {X 0,Y 44.017,Z 937.169,A -85,B 0,C 180,E1 -30121.362,E2 -30121.362} C_VEL
LIN {X 0,Y 39.661,Z 938.723,A -85,B 0,C 180,E1 -30139.775,E2 -30139.775} C_VEL
LIN {X 0,Y 39.166,Z 938.931,A -85,B 0,C 180,E1 -30149.982,E2 -30149.982} C_VEL
LIN {X 0,Y 41.295,Z 938.182,A -85,B 0,C 180,E1 -30169.881,E2 -30169.881} C_VEL
LIN {X 0,Y 43.999,Z 937.232,A -85,B 0,C 180,E1 -30178.614,E2 -30178.614} C_VEL
LIN {X 0,Y 47.413,Z 935.92,A -85,B 0,C 180,E1 -30186.345,E2 -30186.345} C_VEL
LIN {X 0,Y 53.785,Z 933.128,A -85,B 0,C 180,E1 -30195.925,E2 -30195.925} C_VEL
LIN {X 0,Y 61.464,Z 929.272,A -85,B 0,C 180,E1 -30203.147,E2 -30203.147} C_VEL
LIN {X 0,Y 69.726,Z 924.333,A -85,B 0,C 180,E1 -30208.932,E2 -30208.932} C_VEL
LIN {X 0,Y 75.688,Z 920.155,A -85,B 0,C 180,E1 -30212.336,E2 -30212.336} C_VEL
LIN {X 0,Y 77.444,Z 918.448,A -85,B 0,C 180,E1 -30215.137,E2 -30215.137} C_VEL
LIN {X 0,Y 78.572,Z 916.924,A -85,B 0,C 180,E1 -30219.035,E2 -30219.035} C_VEL
LIN {X 0,Y 79.2,Z 915.952,A -85,B 0,C 180,E1 -30222.306,E2 -30222.306} C_VEL
LIN {X 0,Y 79.314,Z 915.602,A -85,B 0,C 180,E1 -30225.105,E2 -30225.105} C_VEL
LIN {X 0,Y 78.719,Z 915.929,A -85,B 0,C 180,E1 -30227.934,E2 -30227.934} C_VEL
LIN {X 0,Y 76.336,Z 918.292,A -85,B 0,C 180,E1 -30236.762,E2 -30236.762} C_VEL
LIN {X 0,Y 76.318,Z 918.456,A -85,B 0,C 180,E1 -30237.796,E2 -30237.796} C_VEL
LIN {X 0,Y 76.442,Z 918.748,A -85,B 0,C 180,E1 -30240,E2 -30240} C_VEL
